LIN {X 0,Y 301.093,Z 516.104,A -85,B 0,C 180,E1 -16309.074,E2 -16309.074} C_VEL
LIN {X 0,Y 303.316,Z 506.78,A -85,B 0,C 180,E1 -16311.404,E2 -16311.404} C_VEL
LIN {X 0,Y 305.446,Z 497.307,A -85,B 0,C 180,E1 -16313.385,E2 -16313.385} C_VEL
LIN {X 0,Y 308.235,Z 485.037,A -85,B 0,C 180,E1 -16315.491,E2 -16315.491} C_VEL
LIN {X 0,Y 310.983,Z 472.541,A -85,B 0,C 180,E1 -16317.235,E2 -16317.235} C_VEL
LIN {X 0,Y 313.672,Z 459.222,A -85,B 0,C 180,E1 -16318.741,E2 -16318.741} C_VEL
LIN {X 0,Y 314.374,Z 455.035,A -85,B 0,C 180,E1 -16319.152,E2 -16319.152} C_VEL
LIN {X 0,Y 313.209,Z 443.277,A -85,B 0,C 180,E1 -16320.482,E2 -16320.482} C_VEL
LIN {X 0,Y 311.406,Z 431.077,A -85,B 0,C 180,E1 -16321.735,E2 -16321.735} C_VEL
LIN {X 0,Y 307.92,Z 415.559,A -85,B 0,C 180,E1 -16323.194,E2 -16323.194} C_VEL
LIN {X 0,Y 303.433,Z 400.922,A -85,B 0,C 180,E1 -16324.465,E2 -16324.465} C_VEL
LIN {X 0,Y 299.776,Z 390.786,A -85,B 0,C 180,E1 -16325.294,E2 -16325.294} C_VEL
LIN {X 0,Y 299.637,Z 389.858,A -85,B 0,C 180,E1 -16325.364,E2 -16325.364} C_VEL
LIN {X 0,Y 300.45,Z 384.591,A -85,B 0,C 180,E1 -16329.473,E2 -16329.473} C_VEL
LIN {X 0,Y 300.937,Z 380.64,A -85,B 0,C 180,E1 -16332.63,E2 -16332.63} C_VEL
LIN {X 0,Y 300.629,Z 377.385,A -85,B 0,C 180,E1 -16335.466,E2 -16335.466} C_VEL
LIN {X 0,Y 300.054,Z 373.593,A -85,B 0,C 180,E1 -16339.018,E2 -16339.018} C_VEL
LIN {X 0,Y 299.471,Z 370.212,A -85,B 0,C 180,E1 -16342.399,E2 -16342.399} C_VEL
LIN {X 0,Y 298.977,Z 367.207,A -85,B 0,C 180,E1 -16345.656,E2 -16345.656} C_VEL
LIN {X 0,Y 298.549,Z 364.477,A -85,B 0,C 180,E1 -16348.809,E2 -16348.809} C_VEL
LIN {X 0,Y 298.429,Z 363.938,A -85,B 0,C 180,E1 -16350.617,E2 -16350.617} C_VEL
LIN {X 0,Y 298.485,Z 363.932,A -85,B 0,C 180,E1 -16353.475,E2 -16353.475} C_VEL
LIN {X 0,Y 298.438,Z 363.938,A -85,B 0,C 180,E1 -16356.698,E2 -16356.698} C_VEL
LIN {X 0,Y 298.543,Z 363.922,A -85,B 0,C 180,E1 -16360.757,E2 -16360.757} C_VEL
LIN {X 0,Y 298.597,Z 363.92,A -85,B 0,C 180,E1 -16364.995,E2 -16364.995} C_VEL
LIN {X 0,Y 298.597,Z 363.922,A -85,B 0,C 180,E1 -16369.147,E2 -16369.147} C_VEL
LIN {X 0,Y 298.762,Z 363.898,A -85,B 0,C 180,E1 -16371.886,E2 -16371.886} C_VEL
LIN {X 0,Y 298.664,Z 363.908,A -85,B 0,C 180,E1 -16374.599,E2 -16374.599} C_VEL
LIN {X 0,Y 298.926,Z 363.874,A -85,B 0,C 180,E1 -16378.653,E2 -16378.653} C_VEL
LIN {X 0,Y 298.927,Z 363.876,A -85,B 0,C 180,E1 -16381.347,E2 -16381.347} C_VEL
LIN {X 0,Y 298.802,Z 363.885,A -85,B 0,C 180,E1 -16386.754,E2 -16386.754} C_VEL
LIN {X 0,Y 298.684,Z 363.904,A -85,B 0,C 180,E1 -16389.48,E2 -16389.48} C_VEL
LIN {X 0,Y 298.555,Z 363.892,A -85,B 0,C 180,E1 -16393.615,E2 -16393.615} C_VEL
LIN {X 0,Y 298.552,Z 363.921,A -85,B 0,C 180,E1 -16396.409,E2 -16396.409} C_VEL
LIN {X 0,Y 298.501,Z 363.902,A -85,B 0,C 180,E1 -16399.647,E2 -16399.647} C_VEL
LIN {X 0,Y 298.432,Z 363.935,A -85,B 0,C 180,E1 -16403.6,E2 -16403.6} C_VEL
LIN {X 0,Y 298.49,Z 363.909,A -85,B 0,C 180,E1 -16406.575,E2 -16406.575} C_VEL
LIN {X 0,Y 298.42,Z 363.936,A -85,B 0,C 180,E1 -16409.641,E2 -16409.641} C_VEL
LIN {X 0,Y 298.398,Z 363.924,A -85,B 0,C 180,E1 -16412.8,E2 -16412.8} C_VEL
LIN {X 0,Y 298.467,Z 363.933,A -85,B 0,C 180,E1 -16416.812,E2 -16416.812} C_VEL
LIN {X 0,Y 298.39,Z 363.942,A -85,B 0,C 180,E1 -16421.087,E2 -16421.087} C_VEL
LIN {X 0,Y 298.401,Z 363.942,A -85,B 0,C 180,E1 -16423.103,E2 -16423.103} C_VEL
LIN {X 0,Y 298.341,Z 363.954,A -85,B 0,C 180,E1 -16426.909,E2 -16426.909} C_VEL
LIN {X 0,Y 298.249,Z 363.963,A -85,B 0,C 180,E1 -16428.943,E2 -16428.943} C_VEL
LIN {X 0,Y 298.148,Z 365.832,A -85,B 0,C 180,E1 -16432.202,E2 -16432.202} C_VEL
LIN {X 0,Y 298.084,Z 367.347,A -85,B 0,C 180,E1 -16434.524,E2 -16434.524} C_VEL
LIN {X 0,Y 299.159,Z 370.435,A -85,B 0,C 180,E1 -16434.787,E2 -16434.787} C_VEL
LIN {X 0,Y 300.414,Z 372.767,A -85,B 0,C 180,E1 -16435.038,E2 -16435.038} C_VEL
LIN {X 0,Y 305.803,Z 384.256,A -85,B 0,C 180,E1 -16436.253,E2 -16436.253} C_VEL
LIN {X 0,Y 310.82,Z 397.125,A -85,B 0,C 180,E1 -16437.646,E2 -16437.646} C_VEL
LIN {X 0,Y 314.659,Z 409.849,A -85,B 0,C 180,E1 -16439.088,E2 -16439.088} C_VEL
LIN {X 0,Y 317.153,Z 421.115,A -85,B 0,C 180,E1 -16440.431,E2 -16440.431} C_VEL
LIN {X 0,Y 314.958,Z 434.259,A -85,B 0,C 180,E1 -16441.694,E2 -16441.694} C_VEL
LIN {X 0,Y 312.497,Z 447.415,A -85,B 0,C 180,E1 -16443.269,E2 -16443.269} C_VEL
LIN {X 0,Y 310.041,Z 458.721,A -85,B 0,C 180,E1 -16444.902,E2 -16444.902} C_VEL
LIN {X 0,Y 307.626,Z 469.495,A -85,B 0,C 180,E1 -16446.79,E2 -16446.79} C_VEL
LIN {X 0,Y 305.011,Z 480.245,A -85,B 0,C 180,E1 -16449.074,E2 -16449.074} C_VEL
LIN {X 0,Y 302.818,Z 489.159,A -85,B 0,C 180,E1 -16451.39,E2 -16451.39} C_VEL
LIN {X 0,Y 301.057,Z 496.534,A -85,B 0,C 180,E1 -16453.731,E2 -16453.731} C_VEL
LIN {X 0,Y 299.789,Z 501.835,A -85,B 0,C 180,E1 -16455.749,E2 -16455.749} C_VEL
LIN {X 0,Y 298.494,Z 507.611,A -85,B 0,C 180,E1 -16458.455,E2 -16458.455} C_VEL
LIN {X 0,Y 297.82,Z 511.025,A -85,B 0,C 180,E1 -16460.491,E2 -16460.491} C_VEL
LIN {X 0,Y 297.207,Z 514.571,A -85,B 0,C 180,E1 -16463.299,E2 -16463.299} C_VEL
LIN {X 0,Y 296.882,Z 516.759,A -85,B 0,C 180,E1 -16465.927,E2 -16465.927} C_VEL
LIN {X 0,Y 296.726,Z 517.922,A -85,B 0,C 180,E1 -16468.642,E2 -16468.642} C_VEL
LIN {X 0,Y 296.726,Z 517.935,A -85,B 0,C 180,E1 -16471.357,E2 -16471.357} C_VEL
LIN {X 0,Y 296.881,Z 516.827,A -85,B 0,C 180,E1 -16474.072,E2 -16474.072} C_VEL
LIN {X 0,Y 297.22,Z 514.599,A -85,B 0,C 180,E1 -16476.789,E2 -16476.789} C_VEL
LIN {X 0,Y 297.8,Z 511.195,A -85,B 0,C 180,E1 -16479.508,E2 -16479.508} C_VEL
LIN {X 0,Y 298.741,Z 506.528,A -85,B 0,C 180,E1 -16482.223,E2 -16482.223} C_VEL
LIN {X 0,Y 300.182,Z 500.468,A -85,B 0,C 180,E1 -16484.923,E2 -16484.923} C_VEL
LIN {X 0,Y 301.908,Z 492.838,A -85,B 0,C 180,E1 -16487.615,E2 -16487.615} C_VEL
LIN {X 0,Y 303.968,Z 484.686,A -85,B 0,C 180,E1 -16489.939,E2 -16489.939} C_VEL
LIN {X 0,Y 306.359,Z 474.857,A -85,B 0,C 180,E1 -16492.241,E2 -16492.241} C_VEL
LIN {X 0,Y 308.851,Z 464.107,A -85,B 0,C 180,E1 -16494.313,E2 -16494.313} C_VEL
LIN {X 0,Y 311.593,Z 451.648,A -85,B 0,C 180,E1 -16496.272,E2 -16496.272} C_VEL
LIN {X 0,Y 314.095,Z 439.396,A -85,B 0,C 180,E1 -16497.845,E2 -16497.845} C_VEL
LIN {X 0,Y 316.491,Z 425.99,A -85,B 0,C 180,E1 -16499.243,E2 -16499.243} C_VEL
LIN {X 0,Y 317.131,Z 420.255,A -85,B 0,C 180,E1 -16499.778,E2 -16499.778} C_VEL
LIN {X 0,Y 313.848,Z 406.769,A -85,B 0,C 180,E1 -16501.38,E2 -16501.38} C_VEL
LIN {X 0,Y 309.302,Z 392.975,A -85,B 0,C 180,E1 -16502.922,E2 -16502.922} C_VEL
LIN {X 0,Y 304.052,Z 380.298,A -85,B 0,C 180,E1 -16504.287,E2 -16504.287} C_VEL
LIN {X 0,Y 299.306,Z 370.651,A -85,B 0,C 180,E1 -16505.308,E2 -16505.308} C_VEL
LIN {X 0,Y 298.144,Z 367.656,A -85,B 0,C 180,E1 -16505.572,E2 -16505.572} C_VEL
LIN {X 0,Y 298.082,Z 367.317,A -85,B 0,C 180,E1 -16505.633,E2 -16505.633} C_VEL
LIN {X 0,Y 298.21,Z 364.814,A -85,B 0,C 180,E1 -16509.517,E2 -16509.517} C_VEL
LIN {X 0,Y 298.257,Z 363.953,A -85,B 0,C 180,E1 -16511.282,E2 -16511.282} C_VEL
LIN {X 0,Y 298.352,Z 363.946,A -85,B 0,C 180,E1 -16515.034,E2 -16515.034} C_VEL
LIN {X 0,Y 298.383,Z 363.944,A -85,B 0,C 180,E1 -16518.738,E2 -16518.738} C_VEL
LIN {X 0,Y 298.43,Z 363.938,A -85,B 0,C 180,E1 -16522.244,E2 -16522.244} C_VEL
LIN {X 0,Y 298.407,Z 363.933,A -85,B 0,C 180,E1 -16525.581,E2 -16525.581} C_VEL
LIN {X 0,Y 298.394,Z 363.938,A -85,B 0,C 180,E1 -16528.791,E2 -16528.791} C_VEL
LIN {X 0,Y 298.462,Z 363.917,A -85,B 0,C 180,E1 -16531.904,E2 -16531.904} C_VEL
LIN {X 0,Y 298.484,Z 363.925,A -85,B 0,C 180,E1 -16534.924,E2 -16534.924} C_VEL
LIN {X 0,Y 298.447,Z 363.908,A -85,B 0,C 180,E1 -16539.315,E2 -16539.315} C_VEL
LIN {X 0,Y 298.536,Z 363.92,A -85,B 0,C 180,E1 -16542.179,E2 -16542.179} C_VEL
LIN {X 0,Y 298.591,Z 363.905,A -85,B 0,C 180,E1 -16544.994,E2 -16544.994} C_VEL
LIN {X 0,Y 298.55,Z 363.895,A -85,B 0,C 180,E1 -16546.352,E2 -16546.352} C_VEL
LIN {X 0,Y 297.926,Z 363.976,A -85,B 0,C 180,E1 -16547.479,E2 -16547.479} C_VEL
LIN {X 0,Y 295.141,Z 364.34,A -85,B 0,C 180,E1 -16549.316,E2 -16549.316} C_VEL
LIN {X 0,Y 292.774,Z 364.642,A -85,B 0,C 180,E1 -16550.807,E2 -16550.807} C_VEL
LIN {X 0,Y 291.775,Z 364.763,A -85,B 0,C 180,E1 -16551.96,E2 -16551.96} C_VEL
LIN {X 0,Y 291.703,Z 364.771,A -85,B 0,C 180,E1 -16552.351,E2 -16552.351} C_VEL
LIN {X 0,Y 291.788,Z 364.767,A -85,B 0,C 180,E1 -16557.239,E2 -16557.239} C_VEL
LIN {X 0,Y 291.977,Z 364.743,A -85,B 0,C 180,E1 -16560,E2 -16560} C_VEL
LIN {X 0,Y 291.789,Z 364.764,A -85,B 0,C 180,E1 -16562.761,E2 -16562.761} C_VEL
LIN {X 0,Y 291.744,Z 364.77,A -85,B 0,C 180,E1 -16566.918,E2 -16566.918} C_VEL
LIN {X 0,Y 291.627,Z 364.784,A -85,B 0,C 180,E1 -16569.712,E2 -16569.712} C_VEL
LIN {X 0,Y 291.519,Z 364.798,A -85,B 0,C 180,E1 -16573.95,E2 -16573.95} C_VEL
LIN {X 0,Y 291.485,Z 364.801,A -85,B 0,C 180,E1 -16576.818,E2 -16576.818} C_VEL
LIN {X 0,Y 291.448,Z 364.807,A -85,B 0,C 180,E1 -16579.875,E2 -16579.875} C_VEL
LIN {X 0,Y 291.398,Z 364.816,A -85,B 0,C 180,E1 -16584.205,E2 -16584.205} C_VEL
LIN {X 0,Y 291.42,Z 364.813,A -85,B 0,C 180,E1 -16587.272,E2 -16587.272} C_VEL
LIN {X 0,Y 291.385,Z 364.86,A -85,B 0,C 180,E1 -16589.74,E2 -16589.74} C_VEL
LIN {X 0,Y 291.902,Z 368.045,A -85,B 0,C 180,E1 -16593.625,E2 -16593.625} C_VEL
LIN {X 0,Y 292.474,Z 371.514,A -85,B 0,C 180,E1 -16597.537,E2 -16597.537} C_VEL
LIN {X 0,Y 292.975,Z 374.262,A -85,B 0,C 180,E1 -16600.367,E2 -16600.367} C_VEL
LIN {X 0,Y 293.546,Z 378.133,A -85,B 0,C 180,E1 -16604.091,E2 -16604.091} C_VEL
LIN {X 0,Y 293.914,Z 381.424,A -85,B 0,C 180,E1 -16607.042,E2 -16607.042} C_VEL
LIN {X 0,Y 293.528,Z 384.953,A -85,B 0,C 180,E1 -16610.012,E2 -16610.012} C_VEL
LIN {X 0,Y 292.75,Z 389.496,A -85,B 0,C 180,E1 -16613.667,E2 -16613.667} C_VEL
LIN {X 0,Y 293.745,Z 392.872,A -85,B 0,C 180,E1 -16613.917,E2 -16613.917} C_VEL
LIN {X 0,Y 298.154,Z 404.831,A -85,B 0,C 180,E1 -16614.994,E2 -16614.994} C_VEL
LIN {X 0,Y 302.141,Z 418.676,A -85,B 0,C 180,E1 -16616.283,E2 -16616.283} C_VEL
LIN {X 0,Y 305.296,Z 433.414,A -85,B 0,C 180,E1 -16617.756,E2 -16617.756} C_VEL
LIN {X 0,Y 307.228,Z 447.699,A -85,B 0,C 180,E1 -16619.314,E2 -16619.314} C_VEL
LIN {X 0,Y 307.893,Z 456.22,A -85,B 0,C 180,E1 -16620.329,E2 -16620.329} C_VEL
LIN {X 0,Y 305.201,Z 469.763,A -85,B 0,C 180,E1 -16621.832,E2 -16621.832} C_VEL
LIN {X 0,Y 302.549,Z 481.597,A -85,B 0,C 180,E1 -16623.439,E2 -16623.439} C_VEL
LIN {X 0,Y 300.146,Z 491.697,A -85,B 0,C 180,E1 -16625.073,E2 -16625.073} C_VEL
LIN {X 0,Y 297.432,Z 502.993,A -85,B 0,C 180,E1 -16627.292,E2 -16627.292} C_VEL
LIN {X 0,Y 295.325,Z 512.081,A -85,B 0,C 180,E1 -16629.451,E2 -16629.451} C_VEL
LIN {X 0,Y 293.288,Z 520.461,A -85,B 0,C 180,E1 -16631.85,E2 -16631.85} C_VEL
LIN {X 0,Y 291.593,Z 528.35,A -85,B 0,C 180,E1 -16634.626,E2 -16634.626} C_VEL
LIN {X 0,Y 290.489,Z 534.643,A -85,B 0,C 180,E1 -16637.424,E2 -16637.424} C_VEL
LIN {X 0,Y 289.783,Z 539.519,A -85,B 0,C 180,E1 -16640.226,E2 -16640.226} C_VEL
LIN {X 0,Y 289.55,Z 543.105,A -85,B 0,C 180,E1 -16643.03,E2 -16643.03} C_VEL
LIN {X 0,Y 289.515,Z 545.468,A -85,B 0,C 180,E1 -16645.824,E2 -16645.824} C_VEL
LIN {X 0,Y 289.53,Z 546.656,A -85,B 0,C 180,E1 -16648.61,E2 -16648.61} C_VEL
LIN {X 0,Y 289.581,Z 546.815,A -85,B 0,C 180,E1 -16650.001,E2 -16650.001} C_VEL
LIN {X 0,Y 289.524,Z 546.197,A -85,B 0,C 180,E1 -16652.783,E2 -16652.783} C_VEL
LIN {X 0,Y 289.586,Z 544.299,A -85,B 0,C 180,E1 -16655.713,E2 -16655.713} C_VEL
LIN {X 0,Y 289.627,Z 541.438,A -85,B 0,C 180,E1 -16658.372,E2 -16658.372} C_VEL
LIN {X 0,Y 290.039,Z 537.211,A -85,B 0,C 180,E1 -16661.178,E2 -16661.178} C_VEL
LIN {X 0,Y 290.979,Z 531.633,A -85,B 0,C 180,E1 -16663.977,E2 -16663.977} C_VEL
LIN {X 0,Y 292.401,Z 524.549,A -85,B 0,C 180,E1 -16666.764,E2 -16666.764} C_VEL
LIN {X 0,Y 294.312,Z 515.75,A -85,B 0,C 180,E1 -16669.531,E2 -16669.531} C_VEL
LIN {X 0,Y 296.621,Z 506.425,A -85,B 0,C 180,E1 -16671.912,E2 -16671.912} C_VEL
LIN {X 0,Y 298.867,Z 496.952,A -85,B 0,C 180,E1 -16673.932,E2 -16673.932} C_VEL
LIN {X 0,Y 301.779,Z 484.683,A -85,B 0,C 180,E1 -16676.077,E2 -16676.077} C_VEL
LIN {X 0,Y 304.616,Z 472.185,A -85,B 0,C 180,E1 -16677.853,E2 -16677.853} C_VEL
LIN {X 0,Y 307.466,Z 458.73,A -85,B 0,C 180,E1 -16679.394,E2 -16679.394} C_VEL
LIN {X 0,Y 307.877,Z 456.13,A -85,B 0,C 180,E1 -16679.657,E2 -16679.657} C_VEL
LIN {X 0,Y 306.607,Z 442.894,A -85,B 0,C 180,E1 -16681.211,E2 -16681.211} C_VEL
LIN {X 0,Y 304.714,Z 430.324,A -85,B 0,C 180,E1 -16682.546,E2 -16682.546} C_VEL
LIN {X 0,Y 301.144,Z 414.784,A -85,B 0,C 180,E1 -16684.064,E2 -16684.064} C_VEL
LIN {X 0,Y 296.174,Z 399.218,A -85,B 0,C 180,E1 -16685.491,E2 -16685.491} C_VEL
LIN {X 0,Y 293.567,Z 392.489,A -85,B 0,C 180,E1 -16686.087,E2 -16686.087} C_VEL
LIN {X 0,Y 292.771,Z 389.434,A -85,B 0,C 180,E1 -16686.339,E2 -16686.339} C_VEL
LIN {X 0,Y 293.539,Z 384.573,A -85,B 0,C 180,E1 -16690.275,E2 -16690.275} C_VEL
LIN {X 0,Y 293.915,Z 381.328,A -85,B 0,C 180,E1 -16692.959,E2 -16692.959} C_VEL
LIN {X 0,Y 293.53,Z 377.943,A -85,B 0,C 180,E1 -16696.025,E2 -16696.025} C_VEL
LIN {X 0,Y 292.945,Z 374.215,A -85,B 0,C 180,E1 -16699.628,E2 -16699.628} C_VEL
LIN {X 0,Y 292.427,Z 370.907,A -85,B 0,C 180,E1 -16703.071,E2 -16703.071} C_VEL
LIN {X 0,Y 291.874,Z 367.974,A -85,B 0,C 180,E1 -16706.371,E2 -16706.371} C_VEL
LIN {X 0,Y 291.386,Z 364.816,A -85,B 0,C 180,E1 -16710.262,E2 -16710.262} C_VEL
LIN {X 0,Y 291.419,Z 364.812,A -85,B 0,C 180,E1 -16714.272,E2 -16714.272} C_VEL
LIN {X 0,Y 291.385,Z 364.815,A -85,B 0,C 180,E1 -16717.3,E2 -16717.3} C_VEL
LIN {X 0,Y 291.462,Z 364.806,A -85,B 0,C 180,E1 -16720.271,E2 -16720.271} C_VEL
LIN {X 0,Y 291.558,Z 364.796,A -85,B 0,C 180,E1 -16724.624,E2 -16724.624} C_VEL
LIN {X 0,Y 291.54,Z 364.799,A -85,B 0,C 180,E1 -16728.881,E2 -16728.881} C_VEL
LIN {X 0,Y 291.713,Z 364.776,A -85,B 0,C 180,E1 -16731.689,E2 -16731.689} C_VEL
LIN {X 0,Y 291.634,Z 364.784,A -85,B 0,C 180,E1 -16734.469,E2 -16734.469} C_VEL
LIN {X 0,Y 291.892,Z 364.751,A -85,B 0,C 180,E1 -16738.62,E2 -16738.62} C_VEL
LIN {X 0,Y 291.894,Z 364.753,A -85,B 0,C 180,E1 -16741.38,E2 -16741.38} C_VEL
LIN {X 0,Y 291.75,Z 364.763,A -85,B 0,C 180,E1 -16746.918,E2 -16746.918} C_VEL
LIN {X 0,Y 291.633,Z 364.782,A -85,B 0,C 180,E1 -16749.712,E2 -16749.712} C_VEL
LIN {X 0,Y 291.525,Z 364.771,A -85,B 0,C 180,E1 -16753.95,E2 -16753.95} C_VEL
LIN {X 0,Y 291.49,Z 364.801,A -85,B 0,C 180,E1 -16756.818,E2 -16756.818} C_VEL
LIN {X 0,Y 291.454,Z 364.777,A -85,B 0,C 180,E1 -16759.875,E2 -16759.875} C_VEL
LIN {X 0,Y 291.387,Z 364.814,A -85,B 0,C 180,E1 -16764.207,E2 -16764.207} C_VEL
LIN {X 0,Y 291.423,Z 364.786,A -85,B 0,C 180,E1 -16767.272,E2 -16767.272} C_VEL
LIN {X 0,Y 291.337,Z 364.821,A -85,B 0,C 180,E1 -16770.437,E2 -16770.437} C_VEL
LIN {X 0,Y 291.348,Z 364.8,A -85,B 0,C 180,E1 -16773.698,E2 -16773.698} C_VEL
LIN {X 0,Y 291.397,Z 364.813,A -85,B 0,C 180,E1 -16777.258,E2 -16777.258} C_VEL
LIN {X 0,Y 291.337,Z 364.823,A -85,B 0,C 180,E1 -16780.642,E2 -16780.642} C_VEL
LIN {X 0,Y 291.293,Z 364.829,A -85,B 0,C 180,E1 -16784.402,E2 -16784.402} C_VEL
LIN {X 0,Y 291.218,Z 364.84,A -85,B 0,C 180,E1 -16788.429,E2 -16788.429} C_VEL
LIN {X 0,Y 291.195,Z 366.217,A -85,B 0,C 180,E1 -16791.133,E2 -16791.133} C_VEL
LIN {X 0,Y 291.077,Z 367.767,A -85,B 0,C 180,E1 -16793.544,E2 -16793.544} C_VEL
LIN {X 0,Y 292.155,Z 370.783,A -85,B 0,C 180,E1 -16793.808,E2 -16793.808} C_VEL
LIN {X 0,Y 293.526,Z 373.281,A -85,B 0,C 180,E1 -16794.095,E2 -16794.095} C_VEL
LIN {X 0,Y 299.644,Z 386.04,A -85,B 0,C 180,E1 -16795.541,E2 -16795.541} C_VEL
LIN {X 0,Y 304.505,Z 398.844,A -85,B 0,C 180,E1 -16796.99,E2 -16796.99} C_VEL
LIN {X 0,Y 308.201,Z 410.948,A -85,B 0,C 180,E1 -16798.428,E2 -16798.428} C_VEL
LIN {X 0,Y 310.796,Z 422.533,A -85,B 0,C 180,E1 -16799.877,E2 -16799.877} C_VEL
LIN {X 0,Y 308.47,Z 436.029,A -85,B 0,C 180,E1 -16801.229,E2 -16801.229} C_VEL
LIN {X 0,Y 305.911,Z 448.932,A -85,B 0,C 180,E1 -16802.831,E2 -16802.831} C_VEL
LIN {X 0,Y 303.238,Z 460.593,A -85,B 0,C 180,E1 -16804.588,E2 -16804.588} C_VEL
LIN {X 0,Y 300.657,Z 471.474,A -85,B 0,C 180,E1 -16806.585,E2 -16806.585} C_VEL
LIN {X 0,Y 298.369,Z 480.597,A -85,B 0,C 180,E1 -16808.586,E2 -16808.586} C_VEL
LIN {X 0,Y 296.077,Z 489.51,A -85,B 0,C 180,E1 -16810.95,E2 -16810.95} C_VEL
LIN {X 0,Y 294.19,Z 496.887,A -85,B 0,C 180,E1 -16813.341,E2 -16813.341} C_VEL
LIN {X 0,Y 292.903,Z 502.185,A -85,B 0,C 180,E1 -16815.407,E2 -16815.407} C_VEL
LIN {X 0,Y 291.536,Z 507.96,A -85,B 0,C 180,E1 -16818.175,E2 -16818.175} C_VEL
LIN {X 0,Y 290.826,Z 511.373,A -85,B 0,C 180,E1 -16820.26,E2 -16820.26} C_VEL
LIN {X 0,Y 290.136,Z 515.078,A -85,B 0,C 180,E1 -16823.291,E2 -16823.291} C_VEL
LIN {X 0,Y 289.821,Z 517.106,A -85,B 0,C 180,E1 -16825.828,E2 -16825.828} C_VEL
LIN {X 0,Y 289.639,Z 518.269,A -85,B 0,C 180,E1 -16828.609,E2 -16828.609} C_VEL
LIN {X 0,Y 289.639,Z 518.283,A -85,B 0,C 180,E1 -16831.39,E2 -16831.39} C_VEL
LIN {X 0,Y 289.82,Z 517.174,A -85,B 0,C 180,E1 -16834.171,E2 -16834.171} C_VEL
LIN {X 0,Y 290.165,Z 514.947,A -85,B 0,C 180,E1 -16836.955,E2 -16836.955} C_VEL
LIN {X 0,Y 290.804,Z 511.542,A -85,B 0,C 180,E1 -16839.739,E2 -16839.739} C_VEL
LIN {X 0,Y 291.796,Z 506.875,A -85,B 0,C 180,E1 -16842.519,E2 -16842.519} C_VEL
LIN {X 0,Y 293.291,Z 500.816,A -85,B 0,C 180,E1 -16845.282,E2 -16845.282} C_VEL
LIN {X 0,Y 295.123,Z 493.185,A -85,B 0,C 180,E1 -16848.033,E2 -16848.033} C_VEL
LIN {X 0,Y 297.278,Z 485.033,A -85,B 0,C 180,E1 -16850.408,E2 -16850.408} C_VEL
LIN {X 0,Y 299.778,Z 475.204,A -85,B 0,C 180,E1 -16852.756,E2 -16852.756} C_VEL
LIN {X 0,Y 302.488,Z 464.055,A -85,B 0,C 180,E1 -16854.936,E2 -16854.936} C_VEL
LIN {X 0,Y 305.233,Z 451.993,A -85,B 0,C 180,E1 -16856.863,E2 -16856.863} C_VEL
LIN {X 0,Y 307.842,Z 439.739,A -85,B 0,C 180,E1 -16858.461,E2 -16858.461} C_VEL
LIN {X 0,Y 310.329,Z 426.332,A -85,B 0,C 180,E1 -16859.882,E2 -16859.882} C_VEL
LIN {X 0,Y 310.808,Z 423.045,A -85,B 0,C 180,E1 -16860.185,E2 -16860.185} C_VEL
LIN {X 0,Y 309.093,Z 414.317,A -85,B 0,C 180,E1 -16861.27,E2 -16861.27} C_VEL
LIN {X 0,Y 305.722,Z 402.495,A -85,B 0,C 180,E1 -16862.697,E2 -16862.697} C_VEL
LIN {X 0,Y 301.143,Z 389.817,A -85,B 0,C 180,E1 -16864.169,E2 -16864.169} C_VEL
LIN {X 0,Y 295.84,Z 377.893,A -85,B 0,C 180,E1 -16865.511,E2 -16865.511} C_VEL
LIN {X 0,Y 292.558,Z 371.39,A -85,B 0,C 180,E1 -16866.237,E2 -16866.237} C_VEL
LIN {X 0,Y 291.302,Z 368.749,A -85,B 0,C 180,E1 -16866.516,E2 -16866.516} C_VEL
LIN {X 0,Y 291.104,Z 367.725,A -85,B 0,C 180,E1 -16866.608,E2 -16866.608} C_VEL
LIN {X 0,Y 291.205,Z 365.953,A -85,B 0,C 180,E1 -16869.439,E2 -16869.439} C_VEL
LIN {X 0,Y 291.214,Z 364.83,A -85,B 0,C 180,E1 -16871.571,E2 -16871.571} C_VEL
LIN {X 0,Y 291.289,Z 364.826,A -85,B 0,C 180,E1 -16875.598,E2 -16875.598} C_VEL
LIN {X 0,Y 291.333,Z 364.821,A -85,B 0,C 180,E1 -16879.357,E2 -16879.357} C_VEL
LIN {X 0,Y 291.423,Z 364.809,A -85,B 0,C 180,E1 -16882.922,E2 -16882.922} C_VEL
LIN {X 0,Y 291.343,Z 364.804,A -85,B 0,C 180,E1 -16886.301,E2 -16886.301} C_VEL
LIN {X 0,Y 291.386,Z 364.813,A -85,B 0,C 180,E1 -16890.26,E2 -16890.26} C_VEL
LIN {X 0,Y 291.415,Z 364.798,A -85,B 0,C 180,E1 -16894.272,E2 -16894.272} C_VEL
LIN {X 0,Y 291.38,Z 364.809,A -85,B 0,C 180,E1 -16897.299,E2 -16897.299} C_VEL
LIN {X 0,Y 291.456,Z 364.781,A -85,B 0,C 180,E1 -16900.27,E2 -16900.27} C_VEL
LIN {X 0,Y 291.553,Z 364.785,A -85,B 0,C 180,E1 -16904.623,E2 -16904.623} C_VEL
LIN {X 0,Y 291.537,Z 364.785,A -85,B 0,C 180,E1 -16908.88,E2 -16908.88} C_VEL
LIN {X 0,Y 291.703,Z 364.771,A -85,B 0,C 180,E1 -16912.351,E2 -16912.351} C_VEL
LIN {X 0,Y 291.053,Z 364.856,A -85,B 0,C 180,E1 -16913.502,E2 -16913.502} C_VEL
LIN {X 0,Y 288.196,Z 365.213,A -85,B 0,C 180,E1 -16915.376,E2 -16915.376} C_VEL
LIN {X 0,Y 285.817,Z 365.508,A -85,B 0,C 180,E1 -16916.898,E2 -16916.898} C_VEL
LIN {X 0,Y 284.873,Z 365.626,A -85,B 0,C 180,E1 -16918.077,E2 -16918.077} C_VEL
LIN {X 0,Y 284.839,Z 365.629,A -85,B 0,C 180,E1 -16918.476,E2 -16918.476} C_VEL
LIN {X 0,Y 284.854,Z 365.63,A -85,B 0,C 180,E1 -16921.414,E2 -16921.414} C_VEL
LIN {X 0,Y 284.696,Z 365.648,A -85,B 0,C 180,E1 -16927.09,E2 -16927.09} C_VEL
LIN {X 0,Y 284.564,Z 365.663,A -85,B 0,C 180,E1 -16929.955,E2 -16929.955} C_VEL
LIN {X 0,Y 284.479,Z 365.674,A -85,B 0,C 180,E1 -16934.303,E2 -16934.303} C_VEL
LIN {X 0,Y 284.423,Z 365.681,A -85,B 0,C 180,E1 -16937.248,E2 -16937.248} C_VEL
LIN {X 0,Y 284.376,Z 365.685,A -85,B 0,C 180,E1 -16940.242,E2 -16940.242} C_VEL
LIN {X 0,Y 284.367,Z 365.691,A -85,B 0,C 180,E1 -16943.876,E2 -16943.876} C_VEL
LIN {X 0,Y 284.395,Z 365.688,A -85,B 0,C 180,E1 -16947.174,E2 -16947.174} C_VEL
LIN {X 0,Y 284.417,Z 366.236,A -85,B 0,C 180,E1 -16949.617,E2 -16949.617} C_VEL
LIN {X 0,Y 284.845,Z 368.875,A -85,B 0,C 180,E1 -16952.979,E2 -16952.979} C_VEL
LIN {X 0,Y 285.307,Z 371.683,A -85,B 0,C 180,E1 -16956.242,E2 -16956.242} C_VEL
LIN {X 0,Y 285.987,Z 375.526,A -85,B 0,C 180,E1 -16960.377,E2 -16960.377} C_VEL
LIN {X 0,Y 286.601,Z 379.899,A -85,B 0,C 180,E1 -16964.674,E2 -16964.674} C_VEL
LIN {X 0,Y 286.865,Z 382.78,A -85,B 0,C 180,E1 -16967.305,E2 -16967.305} C_VEL
LIN {X 0,Y 286.389,Z 386.32,A -85,B 0,C 180,E1 -16970.355,E2 -16970.355} C_VEL
LIN {X 0,Y 285.918,Z 389.064,A -85,B 0,C 180,E1 -16972.637,E2 -16972.637} C_VEL
LIN {X 0,Y 286.878,Z 392.47,A -85,B 0,C 180,E1 -16972.911,E2 -16972.911} C_VEL
LIN {X 0,Y 287.832,Z 394.8,A -85,B 0,C 180,E1 -16973.136,E2 -16973.136} C_VEL
LIN {X 0,Y 292.175,Z 406.787,A -85,B 0,C 180,E1 -16974.278,E2 -16974.278} C_VEL
LIN {X 0,Y 296.225,Z 421.176,A -85,B 0,C 180,E1 -16975.706,E2 -16975.706} C_VEL
LIN {X 0,Y 299.257,Z 436.303,A -85,B 0,C 180,E1 -16977.307,E2 -16977.307} C_VEL
LIN {X 0,Y 300.89,Z 449.869,A -85,B 0,C 180,E1 -16978.871,E2 -16978.871} C_VEL
LIN {X 0,Y 301.417,Z 457.273,A -85,B 0,C 180,E1 -16979.796,E2 -16979.796} C_VEL
LIN {X 0,Y 298.926,Z 469.417,A -85,B 0,C 180,E1 -16981.186,E2 -16981.186} C_VEL
LIN {X 0,Y 295.9,Z 482.326,A -85,B 0,C 180,E1 -16982.984,E2 -16982.984} C_VEL
LIN {X 0,Y 293.193,Z 493.145,A -85,B 0,C 180,E1 -16984.82,E2 -16984.82} C_VEL
LIN {X 0,Y 290.642,Z 503.338,A -85,B 0,C 180,E1 -16986.905,E2 -16986.905} C_VEL
LIN {X 0,Y 288.622,Z 511.731,A -85,B 0,C 180,E1 -16988.952,E2 -16988.952} C_VEL
LIN {X 0,Y 286.463,Z 520.11,A -85,B 0,C 180,E1 -16991.402,E2 -16991.402} C_VEL
LIN {X 0,Y 284.627,Z 528.303,A -85,B 0,C 180,E1 -16994.362,E2 -16994.362} C_VEL
LIN {X 0,Y 283.495,Z 534.293,A -85,B 0,C 180,E1 -16997.109,E2 -16997.109} C_VEL
LIN {X 0,Y 282.73,Z 539.169,A -85,B 0,C 180,E1 -16999.98,E2 -16999.98} C_VEL
LIN {X 0,Y 282.465,Z 542.755,A -85,B 0,C 180,E1 -17002.854,E2 -17002.854} C_VEL
LIN {X 0,Y 282.415,Z 545.119,A -85,B 0,C 180,E1 -17005.719,E2 -17005.719} C_VEL
LIN {X 0,Y 282.447,Z 546.309,A -85,B 0,C 180,E1 -17008.575,E2 -17008.575} C_VEL
LIN {X 0,Y 282.494,Z 546.467,A -85,B 0,C 180,E1 -17010.001,E2 -17010.001} C_VEL
LIN {X 0,Y 282.45,Z 545.85,A -85,B 0,C 180,E1 -17012.853,E2 -17012.853} C_VEL
LIN {X 0,Y 282.487,Z 544.067,A -85,B 0,C 180,E1 -17015.712,E2 -17015.712} C_VEL
LIN {X 0,Y 282.557,Z 541.087,A -85,B 0,C 180,E1 -17018.583,E2 -17018.583} C_VEL
LIN {X 0,Y 283.011,Z 536.859,A -85,B 0,C 180,E1 -17021.459,E2 -17021.459} C_VEL
LIN {X 0,Y 284.02,Z 531.28,A -85,B 0,C 180,E1 -17024.327,E2 -17024.327} C_VEL
LIN {X 0,Y 285.519,Z 524.195,A -85,B 0,C 180,E1 -17027.181,E2 -17027.181} C_VEL
LIN {X 0,Y 287.555,Z 515.396,A -85,B 0,C 180,E1 -17030.01,E2 -17030.01} C_VEL
LIN {X 0,Y 289.96,Z 506.07,A -85,B 0,C 180,E1 -17032.442,E2 -17032.442} C_VEL
LIN {X 0,Y 292.334,Z 496.599,A -85,B 0,C 180,E1 -17034.502,E2 -17034.502} C_VEL
LIN {X 0,Y 295.357,Z 484.328,A -85,B 0,C 180,E1 -17036.688,E2 -17036.688} C_VEL
LIN {X 0,Y 298.345,Z 471.833,A -85,B 0,C 180,E1 -17038.492,E2 -17038.492} C_VEL
LIN {X 0,Y 301.005,Z 459.613,A -85,B 0,C 180,E1 -17039.931,E2 -17039.931} C_VEL
LIN {X 0,Y 301.351,Z 457.667,A -85,B 0,C 180,E1 -17040.136,E2 -17040.136} C_VEL
LIN {X 0,Y 300.396,Z 445.416,A -85,B 0,C 180,E1 -17041.642,E2 -17041.642} C_VEL
LIN {X 0,Y 298.493,Z 432.171,A -85,B 0,C 180,E1 -17043.117,E2 -17043.117} C_VEL
LIN {X 0,Y 295.244,Z 417.409,A -85,B 0,C 180,E1 -17044.642,E2 -17044.642} C_VEL
LIN {X 0,Y 290.815,Z 402.842,A -85,B 0,C 180,E1 -17046.063,E2 -17046.063} C_VEL
LIN {X 0,Y 287.082,Z 392.869,A -85,B 0,C 180,E1 -17047.008,E2 -17047.008} C_VEL
LIN {X 0,Y 286.001,Z 389.931,A -85,B 0,C 180,E1 -17047.271,E2 -17047.271} C_VEL
LIN {X 0,Y 285.911,Z 389.023,A -85,B 0,C 180,E1 -17047.366,E2 -17047.366} C_VEL
LIN {X 0,Y 286.756,Z 384.185,A -85,B 0,C 180,E1 -17051.433,E2 -17051.433} C_VEL
LIN {X 0,Y 286.885,Z 382.013,A -85,B 0,C 180,E1 -17053.31,E2 -17053.31} C_VEL
LIN {X 0,Y 286.406,Z 378.481,A -85,B 0,C 180,E1 -17056.601,E2 -17056.601} C_VEL
LIN {X 0,Y 285.867,Z 374.837,A -85,B 0,C 180,E1 -17060.268,E2 -17060.268} C_VEL
LIN {X 0,Y 285.218,Z 371.049,A -85,B 0,C 180,E1 -17064.406,E2 -17064.406} C_VEL
LIN {X 0,Y 284.588,Z 367.422,A -85,B 0,C 180,E1 -17068.762,E2 -17068.762} C_VEL
LIN {X 0,Y 284.415,Z 366.184,A -85,B 0,C 180,E1 -17070.383,E2 -17070.383} C_VEL
LIN {X 0,Y 284.399,Z 365.686,A -85,B 0,C 180,E1 -17072.827,E2 -17072.827} C_VEL
LIN {X 0,Y 284.369,Z 365.69,A -85,B 0,C 180,E1 -17076.707,E2 -17076.707} C_VEL
LIN {X 0,Y 284.407,Z 365.685,A -85,B 0,C 180,E1 -17081.262,E2 -17081.262} C_VEL
LIN {X 0,Y 284.495,Z 365.676,A -85,B 0,C 180,E1 -17084.459,E2 -17084.459} C_VEL
LIN {X 0,Y 284.492,Z 365.677,A -85,B 0,C 180,E1 -17088.602,E2 -17088.602} C_VEL
LIN {X 0,Y 284.663,Z 365.654,A -85,B 0,C 180,E1 -17091.481,E2 -17091.481} C_VEL
LIN {X 0,Y 284.605,Z 365.659,A -85,B 0,C 180,E1 -17094.331,E2 -17094.331} C_VEL
LIN {X 0,Y 284.858,Z 365.627,A -85,B 0,C 180,E1 -17098.586,E2 -17098.586} C_VEL
LIN {X 0,Y 284.86,Z 365.629,A -85,B 0,C 180,E1 -17101.414,E2 -17101.414} C_VEL
LIN {X 0,Y 284.702,Z 365.641,A -85,B 0,C 180,E1 -17107.09,E2 -17107.09} C_VEL
LIN {X 0,Y 284.57,Z 365.66,A -85,B 0,C 180,E1 -17109.955,E2 -17109.955} C_VEL
LIN {X 0,Y 284.485,Z 365.652,A -85,B 0,C 180,E1 -17114.303,E2 -17114.303} C_VEL
LIN {X 0,Y 284.427,Z 365.679,A -85,B 0,C 180,E1 -17117.248,E2 -17117.248} C_VEL
LIN {X 0,Y 284.381,Z 365.656,A -85,B 0,C 180,E1 -17120.242,E2 -17120.242} C_VEL
LIN {X 0,Y 284.341,Z 365.688,A -85,B 0,C 180,E1 -17124.846,E2 -17124.846} C_VEL
LIN {X 0,Y 284.331,Z 365.672,A -85,B 0,C 180,E1 -17128.011,E2 -17128.011} C_VEL
LIN {X 0,Y 284.297,Z 365.695,A -85,B 0,C 180,E1 -17131.274,E2 -17131.274} C_VEL
LIN {X 0,Y 284.365,Z 365.686,A -85,B 0,C 180,E1 -17135.354,E2 -17135.354} C_VEL
LIN {X 0,Y 284.326,Z 365.695,A -85,B 0,C 180,E1 -17138.167,E2 -17138.167} C_VEL
LIN {X 0,Y 284.272,Z 365.703,A -85,B 0,C 180,E1 -17142.124,E2 -17142.124} C_VEL
LIN {X 0,Y 284.22,Z 365.712,A -85,B 0,C 180,E1 -17146.182,E2 -17146.182} C_VEL
LIN {X 0,Y 284.175,Z 365.718,A -85,B 0,C 180,E1 -17148.106,E2 -17148.106} C_VEL
LIN {X 0,Y 284.169,Z 366.676,A -85,B 0,C 180,E1 -17150.057,E2 -17150.057} C_VEL
LIN {X 0,Y 284.079,Z 368.156,A -85,B 0,C 180,E1 -17152.477,E2 -17152.477} C_VEL
LIN {X 0,Y 285.229,Z 371.291,A -85,B 0,C 180,E1 -17152.786,E2 -17152.786} C_VEL
LIN {X 0,Y 286.426,Z 373.265,A -85,B 0,C 180,E1 -17153.043,E2 -17153.043} C_VEL
LIN {X 0,Y 292.526,Z 385.915,A -85,B 0,C 180,E1 -17154.546,E2 -17154.546} C_VEL
LIN {X 0,Y 297.068,Z 397.186,A -85,B 0,C 180,E1 -17155.897,E2 -17155.897} C_VEL
LIN {X 0,Y 301.193,Z 409.976,A -85,B 0,C 180,E1 -17157.482,E2 -17157.482} C_VEL
LIN {X 0,Y 304.121,Z 422.384,A -85,B 0,C 180,E1 -17159.085,E2 -17159.085} C_VEL
LIN {X 0,Y 304.468,Z 424.418,A -85,B 0,C 180,E1 -17159.351,E2 -17159.351} C_VEL
LIN {X 0,Y 302,Z 437.799,A -85,B 0,C 180,E1 -17160.744,E2 -17160.744} C_VEL
LIN {X 0,Y 299.332,Z 450.45,A -85,B 0,C 180,E1 -17162.373,E2 -17162.373} C_VEL
LIN {X 0,Y 296.4,Z 462.662,A -85,B 0,C 180,E1 -17164.293,E2 -17164.293} C_VEL
LIN {X 0,Y 293.727,Z 473.436,A -85,B 0,C 180,E1 -17166.373,E2 -17166.373} C_VEL
LIN {X 0,Y 291.027,Z 483.624,A -85,B 0,C 180,E1 -17168.762,E2 -17168.762} C_VEL
LIN {X 0,Y 288.731,Z 492.074,A -85,B 0,C 180,E1 -17171.184,E2 -17171.184} C_VEL
LIN {X 0,Y 286.921,Z 499.093,A -85,B 0,C 180,E1 -17173.638,E2 -17173.638} C_VEL
LIN {X 0,Y 285.199,Z 505.603,A -85,B 0,C 180,E1 -17176.461,E2 -17176.461} C_VEL
LIN {X 0,Y 284.076,Z 510.678,A -85,B 0,C 180,E1 -17179.306,E2 -17179.306} C_VEL
LIN {X 0,Y 283.386,Z 513.603,A -85,B 0,C 180,E1 -17181.442,E2 -17181.442} C_VEL
LIN {X 0,Y 282.91,Z 516.457,A -85,B 0,C 180,E1 -17184.297,E2 -17184.297} C_VEL
LIN {X 0,Y 282.624,Z 518.173,A -85,B 0,C 180,E1 -17187.149,E2 -17187.149} C_VEL
LIN {X 0,Y 282.541,Z 518.772,A -85,B 0,C 180,E1 -17189.999,E2 -17189.999} C_VEL
LIN {X 0,Y 282.624,Z 518.213,A -85,B 0,C 180,E1 -17192.85,E2 -17192.85} C_VEL
LIN {X 0,Y 282.912,Z 516.55,A -85,B 0,C 180,E1 -17195.702,E2 -17195.702} C_VEL
LIN {X 0,Y 283.381,Z 513.745,A -85,B 0,C 180,E1 -17198.557,E2 -17198.557} C_VEL
LIN {X 0,Y 284.254,Z 509.721,A -85,B 0,C 180,E1 -17201.407,E2 -17201.407} C_VEL
LIN {X 0,Y 285.499,Z 504.381,A -85,B 0,C 180,E1 -17204.25,E2 -17204.25} C_VEL
LIN {X 0,Y 286.889,Z 499.382,A -85,B 0,C 180,E1 -17206.362,E2 -17206.362} C_VEL
LIN {X 0,Y 288.633,Z 492.431,A -85,B 0,C 180,E1 -17208.821,E2 -17208.821} C_VEL
LIN {X 0,Y 290.96,Z 484.047,A -85,B 0,C 180,E1 -17211.242,E2 -17211.242} C_VEL
LIN {X 0,Y 293.621,Z 473.945,A -85,B 0,C 180,E1 -17213.635,E2 -17213.635} C_VEL
LIN {X 0,Y 296.462,Z 462.732,A -85,B 0,C 180,E1 -17215.803,E2 -17215.803} C_VEL
LIN {X 0,Y 299.193,Z 451.171,A -85,B 0,C 180,E1 -17217.64,E2 -17217.64} C_VEL
LIN {X 0,Y 301.609,Z 440.083,A -85,B 0,C 180,E1 -17219.105,E2 -17219.105} C_VEL
LIN {X 0,Y 304.194,Z 426.674,A -85,B 0,C 180,E1 -17220.549,E2 -17220.549} C_VEL
LIN {X 0,Y 304.495,Z 424.172,A -85,B 0,C 180,E1 -17220.792,E2 -17220.792} C_VEL
LIN {X 0,Y 301.751,Z 411.982,A -85,B 0,C 180,E1 -17222.39,E2 -17222.39} C_VEL
LIN {X 0,Y 297.823,Z 399.308,A -85,B 0,C 180,E1 -17223.966,E2 -17223.966} C_VEL
LIN {X 0,Y 292.756,Z 386.438,A -85,B 0,C 180,E1 -17225.515,E2 -17225.515} C_VEL
LIN {X 0,Y 287.35,Z 375.113,A -85,B 0,C 180,E1 -17226.876,E2 -17226.876} C_VEL
LIN {X 0,Y 285.543,Z 371.708,A -85,B 0,C 180,E1 -17227.279,E2 -17227.279} C_VEL
LIN {X 0,Y 284.289,Z 369.019,A -85,B 0,C 180,E1 -17227.574,E2 -17227.574} C_VEL
LIN {X 0,Y 284.099,Z 368.133,A -85,B 0,C 180,E1 -17227.663,E2 -17227.663} C_VEL
LIN {X 0,Y 284.203,Z 366.701,A -85,B 0,C 180,E1 -17230.011,E2 -17230.011} C_VEL
LIN {X 0,Y 284.176,Z 365.707,A -85,B 0,C 180,E1 -17232.103,E2 -17232.103} C_VEL
LIN {X 0,Y 284.254,Z 365.703,A -85,B 0,C 180,E1 -17236.189,E2 -17236.189} C_VEL
LIN {X 0,Y 284.305,Z 365.697,A -85,B 0,C 180,E1 -17240.023,E2 -17240.023} C_VEL
LIN {X 0,Y 284.348,Z 365.69,A -85,B 0,C 180,E1 -17243.616,E2 -17243.616} C_VEL
LIN {X 0,Y 284.306,Z 365.678,A -85,B 0,C 180,E1 -17247.189,E2 -17247.189} C_VEL
LIN {X 0,Y 284.357,Z 365.688,A -85,B 0,C 180,E1 -17250.376,E2 -17250.376} C_VEL
LIN {X 0,Y 284.376,Z 365.667,A -85,B 0,C 180,E1 -17253.586,E2 -17253.586} C_VEL
LIN {X 0,Y 284.365,Z 365.687,A -85,B 0,C 180,E1 -17256.707,E2 -17256.707} C_VEL
LIN {X 0,Y 284.401,Z 365.671,A -85,B 0,C 180,E1 -17261.261,E2 -17261.261} C_VEL
LIN {X 0,Y 284.49,Z 365.667,A -85,B 0,C 180,E1 -17264.459,E2 -17264.459} C_VEL
LIN {X 0,Y 284.488,Z 365.657,A -85,B 0,C 180,E1 -17268.601,E2 -17268.601} C_VEL
LIN {X 0,Y 284.657,Z 365.651,A -85,B 0,C 180,E1 -17271.481,E2 -17271.481} C_VEL
LIN {X 0,Y 284.6,Z 365.659,A -85,B 0,C 180,E1 -17274.331,E2 -17274.331} C_VEL
LIN {X 0,Y 284.839,Z 365.629,A -85,B 0,C 180,E1 -17278.476,E2 -17278.476} C_VEL
LIN {X 0,Y 284.238,Z 365.709,A -85,B 0,C 180,E1 -17279.656,E2 -17279.656} C_VEL
LIN {X 0,Y 282.595,Z 365.917,A -85,B 0,C 180,E1 -17280.811,E2 -17280.811} C_VEL
LIN {X 0,Y 278.641,Z 366.406,A -85,B 0,C 180,E1 -17283.13,E2 -17283.13} C_VEL
LIN {X 0,Y 277.548,Z 366.539,A -85,B 0,C 180,E1 -17284.343,E2 -17284.343} C_VEL
LIN {X 0,Y 277.476,Z 366.546,A -85,B 0,C 180,E1 -17284.754,E2 -17284.754} C_VEL
LIN {X 0,Y 277.651,Z 366.526,A -85,B 0,C 180,E1 -17287.271,E2 -17287.271} C_VEL
LIN {X 0,Y 277.504,Z 366.542,A -85,B 0,C 180,E1 -17290.211,E2 -17290.211} C_VEL
LIN {X 0,Y 277.432,Z 366.551,A -85,B 0,C 180,E1 -17294.674,E2 -17294.674} C_VEL
LIN {X 0,Y 277.342,Z 366.564,A -85,B 0,C 180,E1 -17299.234,E2 -17299.234} C_VEL
LIN {X 0,Y 277.317,Z 366.57,A -85,B 0,C 180,E1 -17304.171,E2 -17304.171} C_VEL
LIN {X 0,Y 277.323,Z 366.569,A -85,B 0,C 180,E1 -17307.506,E2 -17307.506} C_VEL
LIN {X 0,Y 277.336,Z 367.09,A -85,B 0,C 180,E1 -17308.782,E2 -17308.782} C_VEL
LIN {X 0,Y 277.759,Z 369.568,A -85,B 0,C 180,E1 -17312.097,E2 -17312.097} C_VEL
LIN {X 0,Y 278.306,Z 372.869,A -85,B 0,C 180,E1 -17316.092,E2 -17316.092} C_VEL
LIN {X 0,Y 278.759,Z 375.539,A -85,B 0,C 180,E1 -17319.072,E2 -17319.072} C_VEL
LIN {X 0,Y 279.319,Z 379.121,A -85,B 0,C 180,E1 -17322.793,E2 -17322.793} C_VEL
LIN {X 0,Y 279.686,Z 381.653,A -85,B 0,C 180,E1 -17325.285,E2 -17325.285} C_VEL
LIN {X 0,Y 279.844,Z 383.826,A -85,B 0,C 180,E1 -17327.307,E2 -17327.307} C_VEL
LIN {X 0,Y 279.384,Z 386.978,A -85,B 0,C 180,E1 -17330.1,E2 -17330.1} C_VEL
LIN {X 0,Y 279.09,Z 388.859,A -85,B 0,C 180,E1 -17331.581,E2 -17331.581} C_VEL
LIN {X 0,Y 280.106,Z 392.116,A -85,B 0,C 180,E1 -17331.858,E2 -17331.858} C_VEL
LIN {X 0,Y 284.936,Z 404.617,A -85,B 0,C 180,E1 -17333.137,E2 -17333.137} C_VEL
LIN {X 0,Y 289.094,Z 418.814,A -85,B 0,C 180,E1 -17334.602,E2 -17334.602} C_VEL
LIN {X 0,Y 292.123,Z 432.915,A -85,B 0,C 180,E1 -17336.134,E2 -17336.134} C_VEL
LIN {X 0,Y 293.902,Z 445.123,A -85,B 0,C 180,E1 -17337.553,E2 -17337.553} C_VEL
LIN {X 0,Y 294.945,Z 458.471,A -85,B 0,C 180,E1 -17339.255,E2 -17339.255} C_VEL
LIN {X 0,Y 292.087,Z 471.665,A -85,B 0,C 180,E1 -17340.841,E2 -17340.841} C_VEL
LIN {X 0,Y 288.989,Z 484.131,A -85,B 0,C 180,E1 -17342.676,E2 -17342.676} C_VEL
LIN {X 0,Y 285.785,Z 496.368,A -85,B 0,C 180,E1 -17344.9,E2 -17344.9} C_VEL
LIN {X 0,Y 283.005,Z 507.274,A -85,B 0,C 180,E1 -17347.362,E2 -17347.362} C_VEL
LIN {X 0,Y 280.494,Z 516.361,A -85,B 0,C 180,E1 -17349.848,E2 -17349.848} C_VEL
LIN {X 0,Y 278.673,Z 523.92,A -85,B 0,C 180,E1 -17352.385,E2 -17352.385} C_VEL
LIN {X 0,Y 277.074,Z 530.982,A -85,B 0,C 180,E1 -17355.307,E2 -17355.307} C_VEL
LIN {X 0,Y 275.992,Z 536.546,A -85,B 0,C 180,E1 -17358.246,E2 -17358.246} C_VEL
LIN {X 0,Y 275.472,Z 540.768,A -85,B 0,C 180,E1 -17361.195,E2 -17361.195} C_VEL
LIN {X 0,Y 275.347,Z 544.042,A -85,B 0,C 180,E1 -17364.527,E2 -17364.527} C_VEL
LIN {X 0,Y 275.373,Z 545.513,A -85,B 0,C 180,E1 -17367.075,E2 -17367.075} C_VEL
LIN {X 0,Y 275.41,Z 546.12,A -85,B 0,C 180,E1 -17370.001,E2 -17370.001} C_VEL
LIN {X 0,Y 275.377,Z 545.503,A -85,B 0,C 180,E1 -17372.926,E2 -17372.926} C_VEL
LIN {X 0,Y 275.389,Z 543.716,A -85,B 0,C 180,E1 -17375.86,E2 -17375.86} C_VEL
LIN {X 0,Y 275.473,Z 540.735,A -85,B 0,C 180,E1 -17378.806,E2 -17378.806} C_VEL
LIN {X 0,Y 275.994,Z 536.507,A -85,B 0,C 180,E1 -17381.755,E2 -17381.755} C_VEL
LIN {X 0,Y 277.076,Z 530.927,A -85,B 0,C 180,E1 -17384.694,E2 -17384.694} C_VEL
LIN {X 0,Y 278.674,Z 523.842,A -85,B 0,C 180,E1 -17387.616,E2 -17387.616} C_VEL
LIN {X 0,Y 280.815,Z 515.042,A -85,B 0,C 180,E1 -17390.511,E2 -17390.511} C_VEL
LIN {X 0,Y 283.351,Z 505.717,A -85,B 0,C 180,E1 -17392.996,E2 -17392.996} C_VEL
LIN {X 0,Y 285.81,Z 496.244,A -85,B 0,C 180,E1 -17395.099,E2 -17395.099} C_VEL
LIN {X 0,Y 288.974,Z 483.974,A -85,B 0,C 180,E1 -17397.326,E2 -17397.326} C_VEL
LIN {X 0,Y 292.111,Z 471.48,A -85,B 0,C 180,E1 -17399.157,E2 -17399.157} C_VEL
LIN {X 0,Y 294.905,Z 458.377,A -85,B 0,C 180,E1 -17400.732,E2 -17400.732} C_VEL
LIN {X 0,Y 293.879,Z 445.034,A -85,B 0,C 180,E1 -17402.428,E2 -17402.428} C_VEL
LIN {X 0,Y 291.82,Z 431.318,A -85,B 0,C 180,E1 -17404.017,E2 -17404.017} C_VEL
LIN {X 0,Y 288.775,Z 417.753,A -85,B 0,C 180,E1 -17405.482,E2 -17405.482} C_VEL
LIN {X 0,Y 284.593,Z 403.752,A -85,B 0,C 180,E1 -17406.918,E2 -17406.918} C_VEL
LIN {X 0,Y 280.157,Z 392.287,A -85,B 0,C 180,E1 -17408.088,E2 -17408.088} C_VEL
LIN {X 0,Y 279.103,Z 389.078,A -85,B 0,C 180,E1 -17408.369,E2 -17408.369} C_VEL
LIN {X 0,Y 279.055,Z 388.647,A -85,B 0,C 180,E1 -17408.426,E2 -17408.426} C_VEL
LIN {X 0,Y 279.631,Z 385.607,A -85,B 0,C 180,E1 -17411.063,E2 -17411.063} C_VEL
LIN {X 0,Y 279.862,Z 383.164,A -85,B 0,C 180,E1 -17413.26,E2 -17413.26} C_VEL
LIN {X 0,Y 279.366,Z 379.384,A -85,B 0,C 180,E1 -17416.85,E2 -17416.85} C_VEL
LIN {X 0,Y 279.035,Z 377.195,A -85,B 0,C 180,E1 -17419.091,E2 -17419.091} C_VEL
LIN {X 0,Y 278.484,Z 373.838,A -85,B 0,C 180,E1 -17422.722,E2 -17422.722} C_VEL
LIN {X 0,Y 277.917,Z 370.578,A -85,B 0,C 180,E1 -17426.566,E2 -17426.566} C_VEL
LIN {X 0,Y 277.569,Z 368.24,A -85,B 0,C 180,E1 -17429.576,E2 -17429.576} C_VEL
LIN {X 0,Y 277.333,Z 367.038,A -85,B 0,C 180,E1 -17431.218,E2 -17431.218} C_VEL
LIN {X 0,Y 277.36,Z 366.562,A -85,B 0,C 180,E1 -17432.864,E2 -17432.864} C_VEL
LIN {X 0,Y 277.332,Z 366.565,A -85,B 0,C 180,E1 -17436.08,E2 -17436.08} C_VEL
LIN {X 0,Y 277.348,Z 366.562,A -85,B 0,C 180,E1 -17440.767,E2 -17440.767} C_VEL
LIN {X 0,Y 277.438,Z 366.556,A -85,B 0,C 180,E1 -17445.326,E2 -17445.326} C_VEL
LIN {X 0,Y 277.51,Z 366.546,A -85,B 0,C 180,E1 -17449.789,E2 -17449.789} C_VEL
LIN {X 0,Y 277.657,Z 366.526,A -85,B 0,C 180,E1 -17452.729,E2 -17452.729} C_VEL
LIN {X 0,Y 277.824,Z 366.503,A -85,B 0,C 180,E1 -17458.551,E2 -17458.551} C_VEL
LIN {X 0,Y 277.825,Z 366.505,A -85,B 0,C 180,E1 -17461.45,E2 -17461.45} C_VEL
LIN {X 0,Y 277.657,Z 366.519,A -85,B 0,C 180,E1 -17467.271,E2 -17467.271} C_VEL
LIN {X 0,Y 277.51,Z 366.535,A -85,B 0,C 180,E1 -17470.211,E2 -17470.211} C_VEL
LIN {X 0,Y 277.438,Z 366.535,A -85,B 0,C 180,E1 -17474.674,E2 -17474.674} C_VEL
LIN {X 0,Y 277.346,Z 366.539,A -85,B 0,C 180,E1 -17479.234,E2 -17479.234} C_VEL
LIN {X 0,Y 277.296,Z 366.569,A -85,B 0,C 180,E1 -17484.158,E2 -17484.158} C_VEL
LIN {X 0,Y 277.327,Z 366.541,A -85,B 0,C 180,E1 -17487.504,E2 -17487.504} C_VEL
LIN {X 0,Y 277.275,Z 366.573,A -85,B 0,C 180,E1 -17490.481,E2 -17490.481} C_VEL
LIN {X 0,Y 277.257,Z 366.555,A -85,B 0,C 180,E1 -17493.895,E2 -17493.895} C_VEL
LIN {X 0,Y 277.284,Z 366.572,A -85,B 0,C 180,E1 -17497.467,E2 -17497.467} C_VEL
LIN {X 0,Y 277.212,Z 366.58,A -85,B 0,C 180,E1 -17501.236,E2 -17501.236} C_VEL
LIN {X 0,Y 277.172,Z 366.591,A -85,B 0,C 180,E1 -17505.233,E2 -17505.233} C_VEL
LIN {X 0,Y 277.135,Z 366.595,A -85,B 0,C 180,E1 -17507.343,E2 -17507.343} C_VEL
LIN {X 0,Y 277.146,Z 367.495,A -85,B 0,C 180,E1 -17509.531,E2 -17509.531} C_VEL
LIN {X 0,Y 277.103,Z 368.667,A -85,B 0,C 180,E1 -17511.379,E2 -17511.379} C_VEL
LIN {X 0,Y 278.207,Z 371.636,A -85,B 0,C 180,E1 -17511.675,E2 -17511.675} C_VEL
LIN {X 0,Y 279.505,Z 373.677,A -85,B 0,C 180,E1 -17511.966,E2 -17511.966} C_VEL
LIN {X 0,Y 285.534,Z 385.971,A -85,B 0,C 180,E1 -17513.518,E2 -17513.518} C_VEL
LIN {X 0,Y 290.375,Z 397.589,A -85,B 0,C 180,E1 -17514.997,E2 -17514.997} C_VEL
LIN {X 0,Y 294.704,Z 411.029,A -85,B 0,C 180,E1 -17516.735,E2 -17516.735} C_VEL
LIN {X 0,Y 297.712,Z 423.573,A -85,B 0,C 180,E1 -17518.436,E2 -17518.436} C_VEL
LIN {X 0,Y 298.055,Z 427.033,A -85,B 0,C 180,E1 -17518.876,E2 -17518.876} C_VEL
LIN {X 0,Y 295.258,Z 440.933,A -85,B 0,C 180,E1 -17520.401,E2 -17520.401} C_VEL
LIN {X 0,Y 292.512,Z 453.124,A -85,B 0,C 180,E1 -17522.061,E2 -17522.061} C_VEL
LIN {X 0,Y 289.491,Z 465.259,A -85,B 0,C 180,E1 -17524.088,E2 -17524.088} C_VEL
LIN {X 0,Y 286.82,Z 475.398,A -85,B 0,C 180,E1 -17526.152,E2 -17526.152} C_VEL
LIN {X 0,Y 284.05,Z 485.312,A -85,B 0,C 180,E1 -17528.595,E2 -17528.595} C_VEL
LIN {X 0,Y 281.708,Z 493.525,A -85,B 0,C 180,E1 -17531.075,E2 -17531.075} C_VEL
LIN {X 0,Y 280.084,Z 499.444,A -85,B 0,C 180,E1 -17533.227,E2 -17533.227} C_VEL
LIN {X 0,Y 278.289,Z 505.953,A -85,B 0,C 180,E1 -17536.118,E2 -17536.118} C_VEL
LIN {X 0,Y 277.073,Z 511.028,A -85,B 0,C 180,E1 -17539.033,E2 -17539.033} C_VEL
LIN {X 0,Y 276.376,Z 513.951,A -85,B 0,C 180,E1 -17541.223,E2 -17541.223} C_VEL
LIN {X 0,Y 275.857,Z 516.805,A -85,B 0,C 180,E1 -17544.15,E2 -17544.15} C_VEL
LIN {X 0,Y 275.553,Z 518.52,A -85,B 0,C 180,E1 -17547.075,E2 -17547.075} C_VEL
LIN {X 0,Y 275.455,Z 519.119,A -85,B 0,C 180,E1 -17549.999,E2 -17549.999} C_VEL
LIN {X 0,Y 275.552,Z 518.56,A -85,B 0,C 180,E1 -17552.923,E2 -17552.923} C_VEL
LIN {X 0,Y 275.858,Z 516.897,A -85,B 0,C 180,E1 -17555.848,E2 -17555.848} C_VEL
LIN {X 0,Y 276.37,Z 514.092,A -85,B 0,C 180,E1 -17558.776,E2 -17558.776} C_VEL
LIN {X 0,Y 277.289,Z 510.069,A -85,B 0,C 180,E1 -17561.698,E2 -17561.698} C_VEL
LIN {X 0,Y 278.611,Z 504.728,A -85,B 0,C 180,E1 -17564.61,E2 -17564.61} C_VEL
LIN {X 0,Y 280.047,Z 499.73,A -85,B 0,C 180,E1 -17566.774,E2 -17566.774} C_VEL
LIN {X 0,Y 281.907,Z 492.778,A -85,B 0,C 180,E1 -17569.288,E2 -17569.288} C_VEL
LIN {X 0,Y 284.35,Z 484.393,A -85,B 0,C 180,E1 -17571.761,E2 -17571.761} C_VEL
LIN {X 0,Y 287.134,Z 474.291,A -85,B 0,C 180,E1 -17574.203,E2 -17574.203} C_VEL
LIN {X 0,Y 289.964,Z 463.537,A -85,B 0,C 180,E1 -17576.334,E2 -17576.334} C_VEL
LIN {X 0,Y 292.655,Z 452.68,A -85,B 0,C 180,E1 -17578.117,E2 -17578.117} C_VEL
LIN {X 0,Y 295.413,Z 440.427,A -85,B 0,C 180,E1 -17579.776,E2 -17579.776} C_VEL
LIN {X 0,Y 298.121,Z 427.015,A -85,B 0,C 180,E1 -17581.24,E2 -17581.24} C_VEL
LIN {X 0,Y 297.94,Z 424.541,A -85,B 0,C 180,E1 -17581.547,E2 -17581.547} C_VEL
LIN {X 0,Y 295.086,Z 412.362,A -85,B 0,C 180,E1 -17583.215,E2 -17583.215} C_VEL
LIN {X 0,Y 291.158,Z 399.802,A -85,B 0,C 180,E1 -17584.845,E2 -17584.845} C_VEL
LIN {X 0,Y 286.137,Z 387.13,A -85,B 0,C 180,E1 -17586.448,E2 -17586.448} C_VEL
LIN {X 0,Y 280.586,Z 375.828,A -85,B 0,C 180,E1 -17587.908,E2 -17587.908} C_VEL
LIN {X 0,Y 278.631,Z 372.219,A -85,B 0,C 180,E1 -17588.365,E2 -17588.365} C_VEL
LIN {X 0,Y 277.27,Z 369.371,A -85,B 0,C 180,E1 -17588.701,E2 -17588.701} C_VEL
LIN {X 0,Y 277.129,Z 368.514,A -85,B 0,C 180,E1 -17588.828,E2 -17588.828} C_VEL
LIN {X 0,Y 277.155,Z 367.113,A -85,B 0,C 180,E1 -17591.245,E2 -17591.245} C_VEL
LIN {X 0,Y 277.142,Z 366.584,A -85,B 0,C 180,E1 -17593.21,E2 -17593.21} C_VEL
LIN {X 0,Y 277.213,Z 366.581,A -85,B 0,C 180,E1 -17597.325,E2 -17597.325} C_VEL
LIN {X 0,Y 277.273,Z 366.572,A -85,B 0,C 180,E1 -17601.789,E2 -17601.789} C_VEL
LIN {X 0,Y 277.302,Z 366.569,A -85,B 0,C 180,E1 -17604.344,E2 -17604.344} C_VEL
LIN {X 0,Y 277.243,Z 366.561,A -85,B 0,C 180,E1 -17607.836,E2 -17607.836} C_VEL
LIN {X 0,Y 277.288,Z 366.561,A -85,B 0,C 180,E1 -17611.212,E2 -17611.212} C_VEL
LIN {X 0,Y 277.312,Z 366.556,A -85,B 0,C 180,E1 -17614.479,E2 -17614.479} C_VEL
LIN {X 0,Y 277.283,Z 366.561,A -85,B 0,C 180,E1 -17617.654,E2 -17617.654} C_VEL
LIN {X 0,Y 277.343,Z 366.542,A -85,B 0,C 180,E1 -17620.766,E2 -17620.766} C_VEL
LIN {X 0,Y 277.433,Z 366.534,A -85,B 0,C 180,E1 -17625.326,E2 -17625.326} C_VEL
LIN {X 0,Y 277.505,Z 366.54,A -85,B 0,C 180,E1 -17629.788,E2 -17629.788} C_VEL
LIN {X 0,Y 277.651,Z 366.526,A -85,B 0,C 180,E1 -17632.729,E2 -17632.729} C_VEL
LIN {X 0,Y 277.82,Z 366.504,A -85,B 0,C 180,E1 -17638.55,E2 -17638.55} C_VEL
LIN {X 0,Y 277.82,Z 366.506,A -85,B 0,C 180,E1 -17641.449,E2 -17641.449} C_VEL
LIN {X 0,Y 277.476,Z 366.546,A -85,B 0,C 180,E1 -17644.754,E2 -17644.754} C_VEL
LIN {X 0,Y 276.852,Z 366.626,A -85,B 0,C 180,E1 -17645.968,E2 -17645.968} C_VEL
LIN {X 0,Y 274.008,Z 366.979,A -85,B 0,C 180,E1 -17647.945,E2 -17647.945} C_VEL
LIN {X 0,Y 271.557,Z 367.284,A -85,B 0,C 180,E1 -17649.552,E2 -17649.552} C_VEL
LIN {X 0,Y 270.488,Z 367.419,A -85,B 0,C 180,E1 -17650.798,E2 -17650.798} C_VEL
LIN {X 0,Y 270.395,Z 367.423,A -85,B 0,C 180,E1 -17651.22,E2 -17651.22} C_VEL
LIN {X 0,Y 270.378,Z 367.425,A -85,B 0,C 180,E1 -17655.901,E2 -17655.901} C_VEL
LIN {X 0,Y 270.29,Z 367.439,A -85,B 0,C 180,E1 -17660.602,E2 -17660.602} C_VEL
LIN {X 0,Y 270.272,Z 367.447,A -85,B 0,C 180,E1 -17664.586,E2 -17664.586} C_VEL
LIN {X 0,Y 270.261,Z 367.449,A -85,B 0,C 180,E1 -17666.236,E2 -17666.236} C_VEL
LIN {X 0,Y 270.317,Z 367.91,A -85,B 0,C 180,E1 -17667.903,E2 -17667.903} C_VEL
LIN {X 0,Y 270.711,Z 370.352,A -85,B 0,C 180,E1 -17671.28,E2 -17671.28} C_VEL
LIN {X 0,Y 271.129,Z 373.097,A -85,B 0,C 180,E1 -17674.769,E2 -17674.769} C_VEL
LIN {X 0,Y 271.778,Z 376.855,A -85,B 0,C 180,E1 -17679.125,E2 -17679.125} C_VEL
LIN {X 0,Y 272.213,Z 379.684,A -85,B 0,C 180,E1 -17682.165,E2 -17682.165} C_VEL
LIN {X 0,Y 272.746,Z 383.67,A -85,B 0,C 180,E1 -17686.177,E2 -17686.177} C_VEL
LIN {X 0,Y 272.656,Z 385.996,A -85,B 0,C 180,E1 -17688.375,E2 -17688.375} C_VEL
LIN {X 0,Y 272.243,Z 388.296,A -85,B 0,C 180,E1 -17690.423,E2 -17690.423} C_VEL
LIN {X 0,Y 273.182,Z 391.529,A -85,B 0,C 180,E1 -17690.701,E2 -17690.701} C_VEL
LIN {X 0,Y 274.466,Z 394.442,A -85,B 0,C 180,E1 -17691.031,E2 -17691.031} C_VEL
LIN {X 0,Y 279.523,Z 408.153,A -85,B 0,C 180,E1 -17692.52,E2 -17692.52} C_VEL
LIN {X 0,Y 283.256,Z 421.318,A -85,B 0,C 180,E1 -17693.963,E2 -17693.963} C_VEL
LIN {X 0,Y 285.869,Z 434.235,A -85,B 0,C 180,E1 -17695.446,E2 -17695.446} C_VEL
LIN {X 0,Y 287.546,Z 446.16,A -85,B 0,C 180,E1 -17696.908,E2 -17696.908} C_VEL
LIN {X 0,Y 288.461,Z 458.287,A -85,B 0,C 180,E1 -17698.51,E2 -17698.51} C_VEL
LIN {X 0,Y 288.176,Z 461.574,A -85,B 0,C 180,E1 -17698.938,E2 -17698.938} C_VEL
LIN {X 0,Y 284.912,Z 474.891,A -85,B 0,C 180,E1 -17700.643,E2 -17700.643} C_VEL
LIN {X 0,Y 281.794,Z 486.766,A -85,B 0,C 180,E1 -17702.524,E2 -17702.524} C_VEL
LIN {X 0,Y 278.865,Z 497.664,A -85,B 0,C 180,E1 -17704.632,E2 -17704.632} C_VEL
LIN {X 0,Y 276.351,Z 506.922,A -85,B 0,C 180,E1 -17706.785,E2 -17706.785} C_VEL
LIN {X 0,Y 273.769,Z 516.011,A -85,B 0,C 180,E1 -17709.331,E2 -17709.331} C_VEL
LIN {X 0,Y 271.816,Z 523.569,A -85,B 0,C 180,E1 -17711.925,E2 -17711.925} C_VEL
LIN {X 0,Y 270.119,Z 530.631,A -85,B 0,C 180,E1 -17714.92,E2 -17714.92} C_VEL
LIN {X 0,Y 268.991,Z 536.197,A -85,B 0,C 180,E1 -17717.936,E2 -17717.936} C_VEL
LIN {X 0,Y 268.409,Z 540.418,A -85,B 0,C 180,E1 -17720.962,E2 -17720.962} C_VEL
LIN {X 0,Y 268.239,Z 543.389,A -85,B 0,C 180,E1 -17723.985,E2 -17723.985} C_VEL
LIN {X 0,Y 268.278,Z 545.165,A -85,B 0,C 180,E1 -17726.997,E2 -17726.997} C_VEL
LIN {X 0,Y 268.328,Z 545.773,A -85,B 0,C 180,E1 -17730.001,E2 -17730.001} C_VEL
LIN {X 0,Y 268.283,Z 545.154,A -85,B 0,C 180,E1 -17733.004,E2 -17733.004} C_VEL
LIN {X 0,Y 268.298,Z 543.367,A -85,B 0,C 180,E1 -17736.015,E2 -17736.015} C_VEL
LIN {X 0,Y 268.41,Z 540.384,A -85,B 0,C 180,E1 -17739.039,E2 -17739.039} C_VEL
LIN {X 0,Y 268.993,Z 536.156,A -85,B 0,C 180,E1 -17742.065,E2 -17742.065} C_VEL
LIN {X 0,Y 270.124,Z 530.573,A -85,B 0,C 180,E1 -17745.081,E2 -17745.081} C_VEL
LIN {X 0,Y 271.818,Z 523.488,A -85,B 0,C 180,E1 -17748.076,E2 -17748.076} C_VEL
LIN {X 0,Y 274.117,Z 514.689,A -85,B 0,C 180,E1 -17751.036,E2 -17751.036} C_VEL
LIN {X 0,Y 276.771,Z 505.364,A -85,B 0,C 180,E1 -17753.575,E2 -17753.575} C_VEL
LIN {X 0,Y 279.322,Z 495.89,A -85,B 0,C 180,E1 -17755.724,E2 -17755.724} C_VEL
LIN {X 0,Y 282.656,Z 483.621,A -85,B 0,C 180,E1 -17757.99,E2 -17757.99} C_VEL
LIN {X 0,Y 285.911,Z 471.127,A -85,B 0,C 180,E1 -17759.853,E2 -17759.853} C_VEL
LIN {X 0,Y 288.443,Z 459.915,A -85,B 0,C 180,E1 -17761.234,E2 -17761.234} C_VEL
LIN {X 0,Y 287.523,Z 446.046,A -85,B 0,C 180,E1 -17763.074,E2 -17763.074} C_VEL
LIN {X 0,Y 285.838,Z 434.009,A -85,B 0,C 180,E1 -17764.545,E2 -17764.545} C_VEL
LIN {X 0,Y 282.874,Z 419.984,A -85,B 0,C 180,E1 -17766.153,E2 -17766.153} C_VEL
LIN {X 0,Y 278.846,Z 406.145,A -85,B 0,C 180,E1 -17767.669,E2 -17767.669} C_VEL
LIN {X 0,Y 273.633,Z 392.42,A -85,B 0,C 180,E1 -17769.144,E2 -17769.144} C_VEL
LIN {X 0,Y 272.384,Z 389.325,A -85,B 0,C 180,E1 -17769.473,E2 -17769.473} C_VEL
LIN {X 0,Y 272.227,Z 388.266,A -85,B 0,C 180,E1 -17769.568,E2 -17769.568} C_VEL
LIN {X 0,Y 272.707,Z 385.467,A -85,B 0,C 180,E1 -17772.072,E2 -17772.072} C_VEL
LIN {X 0,Y 272.772,Z 383.355,A -85,B 0,C 180,E1 -17774.08,E2 -17774.08} C_VEL
LIN {X 0,Y 272.208,Z 379.595,A -85,B 0,C 180,E1 -17777.834,E2 -17777.834} C_VEL
LIN {X 0,Y 271.656,Z 376.074,A -85,B 0,C 180,E1 -17781.618,E2 -17781.618} C_VEL
LIN {X 0,Y 271.013,Z 372.348,A -85,B 0,C 180,E1 -17786.083,E2 -17786.083} C_VEL
LIN {X 0,Y 270.471,Z 369.053,A -85,B 0,C 180,E1 -17790.416,E2 -17790.416} C_VEL
LIN {X 0,Y 270.331,Z 367.838,A -85,B 0,C 180,E1 -17792.12,E2 -17792.12} C_VEL
LIN {X 0,Y 270.266,Z 367.446,A -85,B 0,C 180,E1 -17793.764,E2 -17793.764} C_VEL
LIN {X 0,Y 270.236,Z 367.45,A -85,B 0,C 180,E1 -17797.039,E2 -17797.039} C_VEL
LIN {X 0,Y 270.305,Z 367.441,A -85,B 0,C 180,E1 -17800.245,E2 -17800.245} C_VEL
LIN {X 0,Y 270.406,Z 367.432,A -85,B 0,C 180,E1 -17804.936,E2 -17804.936} C_VEL
LIN {X 0,Y 270.445,Z 367.427,A -85,B 0,C 180,E1 -17809.519,E2 -17809.519} C_VEL
LIN {X 0,Y 270.615,Z 367.404,A -85,B 0,C 180,E1 -17812.539,E2 -17812.539} C_VEL
LIN {X 0,Y 270.79,Z 367.38,A -85,B 0,C 180,E1 -17818.513,E2 -17818.513} C_VEL
LIN {X 0,Y 270.791,Z 367.381,A -85,B 0,C 180,E1 -17821.487,E2 -17821.487} C_VEL
LIN {X 0,Y 270.615,Z 367.396,A -85,B 0,C 180,E1 -17827.461,E2 -17827.461} C_VEL
LIN {X 0,Y 270.445,Z 367.413,A -85,B 0,C 180,E1 -17830.481,E2 -17830.481} C_VEL
LIN {X 0,Y 270.406,Z 367.416,A -85,B 0,C 180,E1 -17835.065,E2 -17835.065} C_VEL
LIN {X 0,Y 270.303,Z 367.41,A -85,B 0,C 180,E1 -17839.756,E2 -17839.756} C_VEL
LIN {X 0,Y 270.241,Z 367.445,A -85,B 0,C 180,E1 -17844.589,E2 -17844.589} C_VEL
LIN {X 0,Y 270.273,Z 367.421,A -85,B 0,C 180,E1 -17847.909,E2 -17847.909} C_VEL
LIN {X 0,Y 270.187,Z 367.451,A -85,B 0,C 180,E1 -17851.348,E2 -17851.348} C_VEL
LIN {X 0,Y 270.218,Z 367.442,A -85,B 0,C 180,E1 -17854.903,E2 -17854.903} C_VEL
LIN {X 0,Y 270.225,Z 367.451,A -85,B 0,C 180,E1 -17858.717,E2 -17858.717} C_VEL
LIN {X 0,Y 270.168,Z 367.459,A -85,B 0,C 180,E1 -17863.249,E2 -17863.249} C_VEL
LIN {X 0,Y 270.099,Z 367.472,A -85,B 0,C 180,E1 -17867.427,E2 -17867.427} C_VEL
LIN {X 0,Y 270.117,Z 368.995,A -85,B 0,C 180,E1 -17870.165,E2 -17870.165} C_VEL
LIN {X 0,Y 271.255,Z 372.073,A -85,B 0,C 180,E1 -17870.504,E2 -17870.504} C_VEL
LIN {X 0,Y 272.717,Z 374.405,A -85,B 0,C 180,E1 -17870.853,E2 -17870.853} C_VEL
LIN {X 0,Y 278.802,Z 386.471,A -85,B 0,C 180,E1 -17872.492,E2 -17872.492} C_VEL
LIN {X 0,Y 283.658,Z 397.898,A -85,B 0,C 180,E1 -17874.034,E2 -17874.034} C_VEL
LIN {X 0,Y 287.581,Z 409.682,A -85,B 0,C 180,E1 -17875.63,E2 -17875.63} C_VEL
LIN {X 0,Y 290.335,Z 420.11,A -85,B 0,C 180,E1 -17877.079,E2 -17877.079} C_VEL
LIN {X 0,Y 291.821,Z 427.458,A -85,B 0,C 180,E1 -17878.141,E2 -17878.141} C_VEL
LIN {X 0,Y 289.391,Z 439.923,A -85,B 0,C 180,E1 -17879.538,E2 -17879.538} C_VEL
LIN {X 0,Y 286.55,Z 452.318,A -85,B 0,C 180,E1 -17881.227,E2 -17881.227} C_VEL
LIN {X 0,Y 283.388,Z 464.373,A -85,B 0,C 180,E1 -17883.227,E2 -17883.227} C_VEL
LIN {X 0,Y 280.769,Z 474.138,A -85,B 0,C 180,E1 -17885.211,E2 -17885.211} C_VEL
LIN {X 0,Y 277.816,Z 484.325,A -85,B 0,C 180,E1 -17887.699,E2 -17887.699} C_VEL
LIN {X 0,Y 275.287,Z 492.776,A -85,B 0,C 180,E1 -17890.228,E2 -17890.228} C_VEL
LIN {X 0,Y 273.259,Z 499.796,A -85,B 0,C 180,E1 -17892.796,E2 -17892.796} C_VEL
LIN {X 0,Y 271.369,Z 506.304,A -85,B 0,C 180,E1 -17895.756,E2 -17895.756} C_VEL
LIN {X 0,Y 270.092,Z 511.378,A -85,B 0,C 180,E1 -17898.746,E2 -17898.746} C_VEL
LIN {X 0,Y 269.344,Z 514.301,A -85,B 0,C 180,E1 -17900.992,E2 -17900.992} C_VEL
LIN {X 0,Y 268.789,Z 517.154,A -85,B 0,C 180,E1 -17903.996,E2 -17903.996} C_VEL
LIN {X 0,Y 268.484,Z 518.868,A -85,B 0,C 180,E1 -17906.998,E2 -17906.998} C_VEL
LIN {X 0,Y 268.372,Z 519.466,A -85,B 0,C 180,E1 -17909.999,E2 -17909.999} C_VEL
LIN {X 0,Y 268.483,Z 518.907,A -85,B 0,C 180,E1 -17913,E2 -17913} C_VEL
LIN {X 0,Y 268.79,Z 517.245,A -85,B 0,C 180,E1 -17916.003,E2 -17916.003} C_VEL
LIN {X 0,Y 269.337,Z 514.44,A -85,B 0,C 180,E1 -17919.007,E2 -17919.007} C_VEL
LIN {X 0,Y 270.336,Z 510.416,A -85,B 0,C 180,E1 -17922.003,E2 -17922.003} C_VEL
LIN {X 0,Y 271.739,Z 505.075,A -85,B 0,C 180,E1 -17924.988,E2 -17924.988} C_VEL
LIN {X 0,Y 273.219,Z 500.079,A -85,B 0,C 180,E1 -17927.206,E2 -17927.206} C_VEL
LIN {X 0,Y 275.192,Z 493.125,A -85,B 0,C 180,E1 -17929.778,E2 -17929.778} C_VEL
LIN {X 0,Y 277.768,Z 484.739,A -85,B 0,C 180,E1 -17932.304,E2 -17932.304} C_VEL
LIN {X 0,Y 280.666,Z 474.636,A -85,B 0,C 180,E1 -17934.798,E2 -17934.798} C_VEL
LIN {X 0,Y 283.722,Z 463.422,A -85,B 0,C 180,E1 -17937.054,E2 -17937.054} C_VEL
LIN {X 0,Y 286.728,Z 451.857,A -85,B 0,C 180,E1 -17938.952,E2 -17938.952} C_VEL
LIN {X 0,Y 289.571,Z 439.366,A -85,B 0,C 180,E1 -17940.642,E2 -17940.642} C_VEL
LIN {X 0,Y 291.755,Z 428.9,A -85,B 0,C 180,E1 -17941.803,E2 -17941.803} C_VEL
LIN {X 0,Y 291.633,Z 426.151,A -85,B 0,C 180,E1 -17942.164,E2 -17942.164} C_VEL
LIN {X 0,Y 288.841,Z 414.001,A -85,B 0,C 180,E1 -17943.9,E2 -17943.9} C_VEL
LIN {X 0,Y 285.076,Z 401.877,A -85,B 0,C 180,E1 -17945.555,E2 -17945.555} C_VEL
LIN {X 0,Y 280.217,Z 389.508,A -85,B 0,C 180,E1 -17947.221,E2 -17947.221} C_VEL
LIN {X 0,Y 274.268,Z 377.195,A -85,B 0,C 180,E1 -17948.897,E2 -17948.897} C_VEL
LIN {X 0,Y 271.929,Z 372.967,A -85,B 0,C 180,E1 -17949.477,E2 -17949.477} C_VEL
LIN {X 0,Y 270.445,Z 370.3,A -85,B 0,C 180,E1 -17949.848,E2 -17949.848} C_VEL
LIN {X 0,Y 270.139,Z 368.974,A -85,B 0,C 180,E1 -17949.96,E2 -17949.96} C_VEL
LIN {X 0,Y 270.096,Z 367.533,A -85,B 0,C 180,E1 -17952.572,E2 -17952.572} C_VEL
LIN {X 0,Y 270.164,Z 367.458,A -85,B 0,C 180,E1 -17956.75,E2 -17956.75} C_VEL
LIN {X 0,Y 270.221,Z 367.449,A -85,B 0,C 180,E1 -17961.282,E2 -17961.282} C_VEL
LIN {X 0,Y 270.213,Z 367.447,A -85,B 0,C 180,E1 -17965.096,E2 -17965.096} C_VEL
LIN {X 0,Y 270.199,Z 367.452,A -85,B 0,C 180,E1 -17969.13,E2 -17969.13} C_VEL
LIN {X 0,Y 270.263,Z 367.424,A -85,B 0,C 180,E1 -17972.145,E2 -17972.145} C_VEL
LIN {X 0,Y 270.275,Z 367.441,A -85,B 0,C 180,E1 -17975.519,E2 -17975.519} C_VEL
LIN {X 0,Y 270.3,Z 367.414,A -85,B 0,C 180,E1 -17980.244,E2 -17980.244} C_VEL
LIN {X 0,Y 270.401,Z 367.415,A -85,B 0,C 180,E1 -17984.935,E2 -17984.935} C_VEL
LIN {X 0,Y 270.44,Z 367.418,A -85,B 0,C 180,E1 -17989.519,E2 -17989.519} C_VEL
LIN {X 0,Y 270.609,Z 367.402,A -85,B 0,C 180,E1 -17992.539,E2 -17992.539} C_VEL
LIN {X 0,Y 270.786,Z 367.38,A -85,B 0,C 180,E1 -17998.513,E2 -17998.513} C_VEL
LIN {X 0,Y 270.786,Z 367.383,A -85,B 0,C 180,E1 -18001.487,E2 -18001.487} C_VEL
LIN {X 0,Y 270.609,Z 367.404,A -85,B 0,C 180,E1 -18007.461,E2 -18007.461} C_VEL
LIN {X 0,Y 270.439,Z 367.423,A -85,B 0,C 180,E1 -18010.481,E2 -18010.481} C_VEL
LIN {X 0,Y 270.395,Z 367.423,A -85,B 0,C 180,E1 -18011.22,E2 -18011.22} C_VEL
LIN {X 0,Y 269.701,Z 367.51,A -85,B 0,C 180,E1 -18012.465,E2 -18012.465} C_VEL
LIN {X 0,Y 266.814,Z 367.874,A -85,B 0,C 180,E1 -18014.491,E2 -18014.491} C_VEL
LIN {X 0,Y 264.371,Z 368.178,A -85,B 0,C 180,E1 -18016.139,E2 -18016.139} C_VEL
LIN {X 0,Y 263.32,Z 368.309,A -85,B 0,C 180,E1 -18017.417,E2 -18017.417} C_VEL
LIN {X 0,Y 263.232,Z 368.316,A -85,B 0,C 180,E1 -18017.85,E2 -18017.85} C_VEL
LIN {X 0,Y 263.215,Z 368.32,A -85,B 0,C 180,E1 -18020.851,E2 -18020.851} C_VEL
LIN {X 0,Y 263.206,Z 368.327,A -85,B 0,C 180,E1 -18025.291,E2 -18025.291} C_VEL
LIN {X 0,Y 263.281,Z 368.771,A -85,B 0,C 180,E1 -18026.987,E2 -18026.987} C_VEL
LIN {X 0,Y 263.784,Z 371.91,A -85,B 0,C 180,E1 -18031.508,E2 -18031.508} C_VEL
LIN {X 0,Y 264.276,Z 375.274,A -85,B 0,C 180,E1 -18035.807,E2 -18035.807} C_VEL
LIN {X 0,Y 264.886,Z 378.591,A -85,B 0,C 180,E1 -18039.698,E2 -18039.698} C_VEL
LIN {X 0,Y 265.41,Z 382.112,A -85,B 0,C 180,E1 -18043.509,E2 -18043.509} C_VEL
LIN {X 0,Y 265.697,Z 385.098,A -85,B 0,C 180,E1 -18046.55,E2 -18046.55} C_VEL
LIN {X 0,Y 265.464,Z 387.948,A -85,B 0,C 180,E1 -18049.206,E2 -18049.206} C_VEL
LIN {X 0,Y 266.395,Z 391.062,A -85,B 0,C 180,E1 -18049.494,E2 -18049.494} C_VEL
LIN {X 0,Y 267.497,Z 393.483,A -85,B 0,C 180,E1 -18049.791,E2 -18049.791} C_VEL
LIN {X 0,Y 272.096,Z 405.341,A -85,B 0,C 180,E1 -18051.161,E2 -18051.161} C_VEL
LIN {X 0,Y 276.231,Z 419.009,A -85,B 0,C 180,E1 -18052.754,E2 -18052.754} C_VEL
LIN {X 0,Y 279.088,Z 431.991,A -85,B 0,C 180,E1 -18054.303,E2 -18054.303} C_VEL
LIN {X 0,Y 281.132,Z 446.006,A -85,B 0,C 180,E1 -18056.078,E2 -18056.078} C_VEL
LIN {X 0,Y 282.051,Z 459.304,A -85,B 0,C 180,E1 -18057.907,E2 -18057.907} C_VEL
LIN {X 0,Y 282.03,Z 461.226,A -85,B 0,C 180,E1 -18058.183,E2 -18058.183} C_VEL
LIN {X 0,Y 278.721,Z 474.545,A -85,B 0,C 180,E1 -18059.925,E2 -18059.925} C_VEL
LIN {X 0,Y 275.467,Z 486.418,A -85,B 0,C 180,E1 -18061.837,E2 -18061.837} C_VEL
LIN {X 0,Y 272.368,Z 497.313,A -85,B 0,C 180,E1 -18063.983,E2 -18063.983} C_VEL
LIN {X 0,Y 269.377,Z 507.948,A -85,B 0,C 180,E1 -18066.557,E2 -18066.557} C_VEL
LIN {X 0,Y 266.714,Z 516.793,A -85,B 0,C 180,E1 -18069.163,E2 -18069.163} C_VEL
LIN {X 0,Y 264.978,Z 523.217,A -85,B 0,C 180,E1 -18071.442,E2 -18071.442} C_VEL
LIN {X 0,Y 263.18,Z 530.28,A -85,B 0,C 180,E1 -18074.512,E2 -18074.512} C_VEL
LIN {X 0,Y 261.998,Z 535.847,A -85,B 0,C 180,E1 -18077.609,E2 -18077.609} C_VEL
LIN {X 0,Y 261.347,Z 540.068,A -85,B 0,C 180,E1 -18080.715,E2 -18080.715} C_VEL
LIN {X 0,Y 261.15,Z 543.04,A -85,B 0,C 180,E1 -18083.821,E2 -18083.821} C_VEL
LIN {X 0,Y 261.185,Z 544.817,A -85,B 0,C 180,E1 -18086.916,E2 -18086.916} C_VEL
LIN {X 0,Y 261.248,Z 545.426,A -85,B 0,C 180,E1 -18090.001,E2 -18090.001} C_VEL
LIN {X 0,Y 261.191,Z 544.806,A -85,B 0,C 180,E1 -18093.086,E2 -18093.086} C_VEL
LIN {X 0,Y 261.217,Z 543.017,A -85,B 0,C 180,E1 -18096.179,E2 -18096.179} C_VEL
LIN {X 0,Y 261.348,Z 540.033,A -85,B 0,C 180,E1 -18099.286,E2 -18099.286} C_VEL
LIN {X 0,Y 262,Z 535.804,A -85,B 0,C 180,E1 -18102.392,E2 -18102.392} C_VEL
LIN {X 0,Y 263.188,Z 530.219,A -85,B 0,C 180,E1 -18105.488,E2 -18105.488} C_VEL
LIN {X 0,Y 264.979,Z 523.133,A -85,B 0,C 180,E1 -18108.559,E2 -18108.559} C_VEL
LIN {X 0,Y 267.079,Z 515.568,A -85,B 0,C 180,E1 -18111.213,E2 -18111.213} C_VEL
LIN {X 0,Y 269.774,Z 506.466,A -85,B 0,C 180,E1 -18113.816,E2 -18113.816} C_VEL
LIN {X 0,Y 272.887,Z 495.536,A -85,B 0,C 180,E1 -18116.377,E2 -18116.377} C_VEL
LIN {X 0,Y 276.34,Z 483.266,A -85,B 0,C 180,E1 -18118.688,E2 -18118.688} C_VEL
LIN {X 0,Y 279.735,Z 470.773,A -85,B 0,C 180,E1 -18120.582,E2 -18120.582} C_VEL
LIN {X 0,Y 282.005,Z 461.078,A -85,B 0,C 180,E1 -18121.808,E2 -18121.808} C_VEL
LIN {X 0,Y 281.332,Z 448.576,A -85,B 0,C 180,E1 -18123.552,E2 -18123.552} C_VEL
LIN {X 0,Y 279.868,Z 436.664,A -85,B 0,C 180,E1 -18125.095,E2 -18125.095} C_VEL
LIN {X 0,Y 277.116,Z 422.818,A -85,B 0,C 180,E1 -18126.77,E2 -18126.77} C_VEL
LIN {X 0,Y 273.136,Z 408.513,A -85,B 0,C 180,E1 -18128.425,E2 -18128.425} C_VEL
LIN {X 0,Y 268.42,Z 395.822,A -85,B 0,C 180,E1 -18129.904,E2 -18129.904} C_VEL
LIN {X 0,Y 266.396,Z 391.141,A -85,B 0,C 180,E1 -18130.455,E2 -18130.455} C_VEL
LIN {X 0,Y 265.421,Z 387.861,A -85,B 0,C 180,E1 -18130.765,E2 -18130.765} C_VEL
LIN {X 0,Y 265.731,Z 385.055,A -85,B 0,C 180,E1 -18133.445,E2 -18133.445} C_VEL
LIN {X 0,Y 265.411,Z 382.062,A -85,B 0,C 180,E1 -18136.491,E2 -18136.491} C_VEL
LIN {X 0,Y 264.828,Z 378.386,A -85,B 0,C 180,E1 -18140.438,E2 -18140.438} C_VEL
LIN {X 0,Y 264.278,Z 375.196,A -85,B 0,C 180,E1 -18144.194,E2 -18144.194} C_VEL
LIN {X 0,Y 263.728,Z 371.847,A -85,B 0,C 180,E1 -18148.514,E2 -18148.514} C_VEL
LIN {X 0,Y 263.259,Z 368.721,A -85,B 0,C 180,E1 -18153.01,E2 -18153.01} C_VEL
LIN {X 0,Y 263.229,Z 368.323,A -85,B 0,C 180,E1 -18155.201,E2 -18155.201} C_VEL
LIN {X 0,Y 263.267,Z 368.317,A -85,B 0,C 180,E1 -18159.694,E2 -18159.694} C_VEL
LIN {X 0,Y 263.354,Z 368.309,A -85,B 0,C 180,E1 -18164.522,E2 -18164.522} C_VEL
LIN {X 0,Y 263.378,Z 368.309,A -85,B 0,C 180,E1 -18169.235,E2 -18169.235} C_VEL
LIN {X 0,Y 263.576,Z 368.282,A -85,B 0,C 180,E1 -18172.339,E2 -18172.339} C_VEL
LIN {X 0,Y 263.755,Z 368.256,A -85,B 0,C 180,E1 -18178.473,E2 -18178.473} C_VEL
LIN {X 0,Y 263.756,Z 368.257,A -85,B 0,C 180,E1 -18181.527,E2 -18181.527} C_VEL
LIN {X 0,Y 263.577,Z 368.274,A -85,B 0,C 180,E1 -18187.662,E2 -18187.662} C_VEL
LIN {X 0,Y 263.378,Z 368.288,A -85,B 0,C 180,E1 -18190.766,E2 -18190.766} C_VEL
LIN {X 0,Y 263.354,Z 368.299,A -85,B 0,C 180,E1 -18195.478,E2 -18195.478} C_VEL
LIN {X 0,Y 263.266,Z 368.284,A -85,B 0,C 180,E1 -18200.307,E2 -18200.307} C_VEL
LIN {X 0,Y 263.196,Z 368.316,A -85,B 0,C 180,E1 -18205.293,E2 -18205.293} C_VEL
LIN {X 0,Y 263.169,Z 368.313,A -85,B 0,C 180,E1 -18208.731,E2 -18208.731} C_VEL
LIN {X 0,Y 263.136,Z 368.318,A -85,B 0,C 180,E1 -18212.288,E2 -18212.288} C_VEL
LIN {X 0,Y 263.191,Z 368.327,A -85,B 0,C 180,E1 -18215.978,E2 -18215.978} C_VEL
LIN {X 0,Y 263.118,Z 368.335,A -85,B 0,C 180,E1 -18219.87,E2 -18219.87} C_VEL
LIN {X 0,Y 263.1,Z 368.343,A -85,B 0,C 180,E1 -18223.989,E2 -18223.989} C_VEL
LIN {X 0,Y 263.064,Z 368.348,A -85,B 0,C 180,E1 -18226.165,E2 -18226.165} C_VEL
LIN {X 0,Y 263.115,Z 369.472,A -85,B 0,C 180,E1 -18228.896,E2 -18228.896} C_VEL
LIN {X 0,Y 264.183,Z 372.296,A -85,B 0,C 180,E1 -18229.217,E2 -18229.217} C_VEL
LIN {X 0,Y 265.813,Z 374.87,A -85,B 0,C 180,E1 -18229.631,E2 -18229.631} C_VEL
LIN {X 0,Y 271.925,Z 386.647,A -85,B 0,C 180,E1 -18231.354,E2 -18231.354} C_VEL
LIN {X 0,Y 276.961,Z 398.236,A -85,B 0,C 180,E1 -18233.015,E2 -18233.015} C_VEL
LIN {X 0,Y 281.043,Z 410.21,A -85,B 0,C 180,E1 -18234.727,E2 -18234.727} C_VEL
LIN {X 0,Y 284.33,Z 423.013,A -85,B 0,C 180,E1 -18236.6,E2 -18236.6} C_VEL
LIN {X 0,Y 285.543,Z 429.943,A -85,B 0,C 180,E1 -18237.639,E2 -18237.639} C_VEL
LIN {X 0,Y 282.718,Z 442.92,A -85,B 0,C 180,E1 -18239.155,E2 -18239.155} C_VEL
LIN {X 0,Y 279.759,Z 454.902,A -85,B 0,C 180,E1 -18240.873,E2 -18240.873} C_VEL
LIN {X 0,Y 276.745,Z 465.963,A -85,B 0,C 180,E1 -18242.798,E2 -18242.798} C_VEL
LIN {X 0,Y 273.862,Z 476.101,A -85,B 0,C 180,E1 -18244.948,E2 -18244.948} C_VEL
LIN {X 0,Y 270.851,Z 486.014,A -85,B 0,C 180,E1 -18247.496,E2 -18247.496} C_VEL
LIN {X 0,Y 268.264,Z 494.228,A -85,B 0,C 180,E1 -18250.087,E2 -18250.087} C_VEL
LIN {X 0,Y 266.459,Z 500.147,A -85,B 0,C 180,E1 -18252.342,E2 -18252.342} C_VEL
LIN {X 0,Y 264.474,Z 506.654,A -85,B 0,C 180,E1 -18255.377,E2 -18255.377} C_VEL
LIN {X 0,Y 263.13,Z 511.727,A -85,B 0,C 180,E1 -18258.444,E2 -18258.444} C_VEL
LIN {X 0,Y 262.32,Z 514.65,A -85,B 0,C 180,E1 -18260.749,E2 -18260.749} C_VEL
LIN {X 0,Y 261.729,Z 517.502,A -85,B 0,C 180,E1 -18263.833,E2 -18263.833} C_VEL
LIN {X 0,Y 261.418,Z 519.215,A -85,B 0,C 180,E1 -18266.917,E2 -18266.917} C_VEL
LIN {X 0,Y 261.292,Z 519.813,A -85,B 0,C 180,E1 -18269.999,E2 -18269.999} C_VEL
LIN {X 0,Y 261.417,Z 519.253,A -85,B 0,C 180,E1 -18273.082,E2 -18273.082} C_VEL
LIN {X 0,Y 261.728,Z 517.592,A -85,B 0,C 180,E1 -18276.165,E2 -18276.165} C_VEL
LIN {X 0,Y 262.311,Z 514.788,A -85,B 0,C 180,E1 -18279.25,E2 -18279.25} C_VEL
LIN {X 0,Y 263.374,Z 510.764,A -85,B 0,C 180,E1 -18282.325,E2 -18282.325} C_VEL
LIN {X 0,Y 264.883,Z 505.422,A -85,B 0,C 180,E1 -18285.386,E2 -18285.386} C_VEL
LIN {X 0,Y 266.41,Z 500.427,A -85,B 0,C 180,E1 -18287.66,E2 -18287.66} C_VEL
LIN {X 0,Y 268.508,Z 493.472,A -85,B 0,C 180,E1 -18290.292,E2 -18290.292} C_VEL
LIN {X 0,Y 271.203,Z 485.085,A -85,B 0,C 180,E1 -18292.874,E2 -18292.874} C_VEL
LIN {X 0,Y 274.218,Z 474.982,A -85,B 0,C 180,E1 -18295.422,E2 -18295.422} C_VEL
LIN {X 0,Y 277.408,Z 463.768,A -85,B 0,C 180,E1 -18297.722,E2 -18297.722} C_VEL
LIN {X 0,Y 280.541,Z 452.201,A -85,B 0,C 180,E1 -18299.654,E2 -18299.654} C_VEL
LIN {X 0,Y 283.5,Z 439.708,A -85,B 0,C 180,E1 -18301.371,E2 -18301.371} C_VEL
LIN {X 0,Y 285.526,Z 430.375,A -85,B 0,C 180,E1 -18302.431,E2 -18302.431} C_VEL
LIN {X 0,Y 285.032,Z 426.253,A -85,B 0,C 180,E1 -18303.035,E2 -18303.035} C_VEL
LIN {X 0,Y 281.935,Z 413.123,A -85,B 0,C 180,E1 -18304.983,E2 -18304.983} C_VEL
LIN {X 0,Y 277.727,Z 400.311,A -85,B 0,C 180,E1 -18306.823,E2 -18306.823} C_VEL
LIN {X 0,Y 272.821,Z 388.496,A -85,B 0,C 180,E1 -18308.505,E2 -18308.505} C_VEL
LIN {X 0,Y 267.148,Z 377.277,A -85,B 0,C 180,E1 -18310.158,E2 -18310.158} C_VEL
LIN {X 0,Y 264.974,Z 373.405,A -85,B 0,C 180,E1 -18310.726,E2 -18310.726} C_VEL
LIN {X 0,Y 263.445,Z 370.673,A -85,B 0,C 180,E1 -18311.133,E2 -18311.133} C_VEL
LIN {X 0,Y 263.125,Z 369.395,A -85,B 0,C 180,E1 -18311.262,E2 -18311.262} C_VEL
LIN {X 0,Y 263.062,Z 368.339,A -85,B 0,C 180,E1 -18313.996,E2 -18313.996} C_VEL
LIN {X 0,Y 263.122,Z 368.335,A -85,B 0,C 180,E1 -18318.106,E2 -18318.106} C_VEL
LIN {X 0,Y 263.164,Z 368.331,A -85,B 0,C 180,E1 -18322.104,E2 -18322.104} C_VEL
LIN {X 0,Y 263.182,Z 368.313,A -85,B 0,C 180,E1 -18325.89,E2 -18325.89} C_VEL
LIN {X 0,Y 263.149,Z 368.331,A -85,B 0,C 180,E1 -18329.506,E2 -18329.506} C_VEL
LIN {X 0,Y 263.191,Z 368.302,A -85,B 0,C 180,E1 -18333.002,E2 -18333.002} C_VEL
LIN {X 0,Y 263.183,Z 368.326,A -85,B 0,C 180,E1 -18336.387,E2 -18336.387} C_VEL
LIN {X 0,Y 263.262,Z 368.288,A -85,B 0,C 180,E1 -18339.693,E2 -18339.693} C_VEL
LIN {X 0,Y 263.349,Z 368.298,A -85,B 0,C 180,E1 -18344.522,E2 -18344.522} C_VEL
LIN {X 0,Y 263.373,Z 368.296,A -85,B 0,C 180,E1 -18349.234,E2 -18349.234} C_VEL
LIN {X 0,Y 263.571,Z 368.278,A -85,B 0,C 180,E1 -18352.338,E2 -18352.338} C_VEL
LIN {X 0,Y 263.75,Z 368.257,A -85,B 0,C 180,E1 -18358.473,E2 -18358.473} C_VEL
LIN {X 0,Y 263.75,Z 368.259,A -85,B 0,C 180,E1 -18361.527,E2 -18361.527} C_VEL
LIN {X 0,Y 263.571,Z 368.28,A -85,B 0,C 180,E1 -18367.661,E2 -18367.661} C_VEL
LIN {X 0,Y 263.372,Z 368.305,A -85,B 0,C 180,E1 -18370.766,E2 -18370.766} C_VEL
LIN {X 0,Y 263.348,Z 368.3,A -85,B 0,C 180,E1 -18375.478,E2 -18375.478} C_VEL
LIN {X 0,Y 263.232,Z 368.316,A -85,B 0,C 180,E1 -18377.85,E2 -18377.85} C_VEL
LIN {X 0,Y 262.552,Z 368.405,A -85,B 0,C 180,E1 -18379.126,E2 -18379.126} C_VEL
LIN {X 0,Y 259.68,Z 368.762,A -85,B 0,C 180,E1 -18381.206,E2 -18381.206} C_VEL
LIN {X 0,Y 257.26,Z 369.068,A -85,B 0,C 180,E1 -18382.897,E2 -18382.897} C_VEL
LIN {X 0,Y 256.24,Z 369.195,A -85,B 0,C 180,E1 -18384.209,E2 -18384.209} C_VEL
LIN {X 0,Y 256.167,Z 369.203,A -85,B 0,C 180,E1 -18384.653,E2 -18384.653} C_VEL
LIN {X 0,Y 256.222,Z 369.636,A -85,B 0,C 180,E1 -18386.032,E2 -18386.032} C_VEL
LIN {X 0,Y 256.563,Z 371.925,A -85,B 0,C 180,E1 -18389.542,E2 -18389.542} C_VEL
LIN {X 0,Y 256.964,Z 374.537,A -85,B 0,C 180,E1 -18393.161,E2 -18393.161} C_VEL
LIN {X 0,Y 257.561,Z 378.12,A -85,B 0,C 180,E1 -18397.693,E2 -18397.693} C_VEL
LIN {X 0,Y 258.022,Z 380.803,A -85,B 0,C 180,E1 -18400.822,E2 -18400.822} C_VEL
LIN {X 0,Y 258.561,Z 384.642,A -85,B 0,C 180,E1 -18405.033,E2 -18405.033} C_VEL
LIN {X 0,Y 258.623,Z 387.467,A -85,B 0,C 180,E1 -18407.882,E2 -18407.882} C_VEL
LIN {X 0,Y 259.599,Z 390.707,A -85,B 0,C 180,E1 -18408.203,E2 -18408.203} C_VEL
LIN {X 0,Y 260.783,Z 392.995,A -85,B 0,C 180,E1 -18408.529,E2 -18408.529} C_VEL
LIN {X 0,Y 265.817,Z 406.069,A -85,B 0,C 180,E1 -18410.135,E2 -18410.135} C_VEL
LIN {X 0,Y 269.615,Z 418.196,A -85,B 0,C 180,E1 -18411.645,E2 -18411.645} C_VEL
LIN {X 0,Y 272.669,Z 431.77,A -85,B 0,C 180,E1 -18413.344,E2 -18413.344} C_VEL
LIN {X 0,Y 274.67,Z 445.34,A -85,B 0,C 180,E1 -18415.131,E2 -18415.131} C_VEL
LIN {X 0,Y 275.566,Z 458.653,A -85,B 0,C 180,E1 -18417.016,E2 -18417.016} C_VEL
LIN {X 0,Y 275.409,Z 463.58,A -85,B 0,C 180,E1 -18417.733,E2 -18417.733} C_VEL
LIN {X 0,Y 271.897,Z 476.558,A -85,B 0,C 180,E1 -18419.519,E2 -18419.519} C_VEL
LIN {X 0,Y 268.593,Z 488.036,A -85,B 0,C 180,E1 -18421.477,E2 -18421.477} C_VEL
LIN {X 0,Y 265.457,Z 498.607,A -85,B 0,C 180,E1 -18423.676,E2 -18423.676} C_VEL
LIN {X 0,Y 262.713,Z 507.763,A -85,B 0,C 180,E1 -18425.977,E2 -18425.977} C_VEL
LIN {X 0,Y 260.036,Z 516.443,A -85,B 0,C 180,E1 -18428.601,E2 -18428.601} C_VEL
LIN {X 0,Y 258.156,Z 522.866,A -85,B 0,C 180,E1 -18430.933,E2 -18430.933} C_VEL
LIN {X 0,Y 256.257,Z 529.928,A -85,B 0,C 180,E1 -18434.083,E2 -18434.083} C_VEL
LIN {X 0,Y 255.013,Z 535.497,A -85,B 0,C 180,E1 -18437.264,E2 -18437.264} C_VEL
LIN {X 0,Y 254.283,Z 539.718,A -85,B 0,C 180,E1 -18440.455,E2 -18440.455} C_VEL
LIN {X 0,Y 254.05,Z 542.69,A -85,B 0,C 180,E1 -18443.648,E2 -18443.648} C_VEL
LIN {X 0,Y 254.096,Z 544.469,A -85,B 0,C 180,E1 -18446.83,E2 -18446.83} C_VEL
LIN {X 0,Y 254.17,Z 545.079,A -85,B 0,C 180,E1 -18450.001,E2 -18450.001} C_VEL
LIN {X 0,Y 254.103,Z 544.458,A -85,B 0,C 180,E1 -18453.172,E2 -18453.172} C_VEL
LIN {X 0,Y 254.14,Z 542.668,A -85,B 0,C 180,E1 -18456.352,E2 -18456.352} C_VEL
LIN {X 0,Y 254.285,Z 539.681,A -85,B 0,C 180,E1 -18459.546,E2 -18459.546} C_VEL
LIN {X 0,Y 255.015,Z 535.452,A -85,B 0,C 180,E1 -18462.737,E2 -18462.737} C_VEL
LIN {X 0,Y 256.265,Z 529.866,A -85,B 0,C 180,E1 -18465.918,E2 -18465.918} C_VEL
LIN {X 0,Y 258.156,Z 522.778,A -85,B 0,C 180,E1 -18469.068,E2 -18469.068} C_VEL
LIN {X 0,Y 260.399,Z 515.214,A -85,B 0,C 180,E1 -18471.784,E2 -18471.784} C_VEL
LIN {X 0,Y 263.169,Z 506.316,A -85,B 0,C 180,E1 -18474.39,E2 -18474.39} C_VEL
LIN {X 0,Y 265.96,Z 496.829,A -85,B 0,C 180,E1 -18476.695,E2 -18476.695} C_VEL
LIN {X 0,Y 269.202,Z 485.911,A -85,B 0,C 180,E1 -18478.881,E2 -18478.881} C_VEL
LIN {X 0,Y 272.577,Z 474.009,A -85,B 0,C 180,E1 -18480.828,E2 -18480.828} C_VEL
LIN {X 0,Y 275.579,Z 462.436,A -85,B 0,C 180,E1 -18482.382,E2 -18482.382} C_VEL
LIN {X 0,Y 275.064,Z 449.982,A -85,B 0,C 180,E1 -18484.202,E2 -18484.202} C_VEL
LIN {X 0,Y 273.341,Z 436.042,A -85,B 0,C 180,E1 -18486.086,E2 -18486.086} C_VEL
LIN {X 0,Y 270.845,Z 423.434,A -85,B 0,C 180,E1 -18487.678,E2 -18487.678} C_VEL
LIN {X 0,Y 267.25,Z 410.412,A -85,B 0,C 180,E1 -18489.284,E2 -18489.284} C_VEL
LIN {X 0,Y 263.18,Z 399.094,A -85,B 0,C 180,E1 -18490.686,E2 -18490.686} C_VEL
LIN {X 0,Y 260.164,Z 391.735,A -85,B 0,C 180,E1 -18491.593,E2 -18491.593} C_VEL
LIN {X 0,Y 258.824,Z 388.563,A -85,B 0,C 180,E1 -18491.986,E2 -18491.986} C_VEL
LIN {X 0,Y 258.62,Z 387.464,A -85,B 0,C 180,E1 -18492.081,E2 -18492.081} C_VEL
LIN {X 0,Y 258.599,Z 384.546,A -85,B 0,C 180,E1 -18495.041,E2 -18495.041} C_VEL
LIN {X 0,Y 258.018,Z 380.732,A -85,B 0,C 180,E1 -18499.177,E2 -18499.177} C_VEL
LIN {X 0,Y 257.462,Z 377.377,A -85,B 0,C 180,E1 -18503.092,E2 -18503.092} C_VEL
LIN {X 0,Y 256.948,Z 374.422,A -85,B 0,C 180,E1 -18506.836,E2 -18506.836} C_VEL
LIN {X 0,Y 256.491,Z 371.318,A -85,B 0,C 180,E1 -18511.262,E2 -18511.262} C_VEL
LIN {X 0,Y 256.191,Z 369.199,A -85,B 0,C 180,E1 -18514.862,E2 -18514.862} C_VEL
LIN {X 0,Y 256.17,Z 369.202,A -85,B 0,C 180,E1 -18519.105,E2 -18519.105} C_VEL
LIN {X 0,Y 256.303,Z 369.188,A -85,B 0,C 180,E1 -18524.085,E2 -18524.085} C_VEL
LIN {X 0,Y 256.313,Z 369.188,A -85,B 0,C 180,E1 -18528.934,E2 -18528.934} C_VEL
LIN {X 0,Y 256.544,Z 369.159,A -85,B 0,C 180,E1 -18532.127,E2 -18532.127} C_VEL
LIN {X 0,Y 256.718,Z 369.133,A -85,B 0,C 180,E1 -18538.431,E2 -18538.431} C_VEL
LIN {X 0,Y 256.718,Z 369.133,A -85,B 0,C 180,E1 -18541.569,E2 -18541.569} C_VEL
LIN {X 0,Y 256.544,Z 369.152,A -85,B 0,C 180,E1 -18547.873,E2 -18547.873} C_VEL
LIN {X 0,Y 256.313,Z 369.161,A -85,B 0,C 180,E1 -18551.066,E2 -18551.066} C_VEL
LIN {X 0,Y 256.304,Z 369.181,A -85,B 0,C 180,E1 -18555.915,E2 -18555.915} C_VEL
LIN {X 0,Y 256.166,Z 369.169,A -85,B 0,C 180,E1 -18560.895,E2 -18560.895} C_VEL
LIN {X 0,Y 256.174,Z 369.193,A -85,B 0,C 180,E1 -18565.13,E2 -18565.13} C_VEL
LIN {X 0,Y 256.107,Z 369.204,A -85,B 0,C 180,E1 -18569.601,E2 -18569.601} C_VEL
LIN {X 0,Y 256.088,Z 369.189,A -85,B 0,C 180,E1 -18573.29,E2 -18573.29} C_VEL
LIN {X 0,Y 256.132,Z 369.206,A -85,B 0,C 180,E1 -18577.275,E2 -18577.275} C_VEL
LIN {X 0,Y 256.06,Z 369.215,A -85,B 0,C 180,E1 -18581.203,E2 -18581.203} C_VEL
LIN {X 0,Y 256.015,Z 369.226,A -85,B 0,C 180,E1 -18585.54,E2 -18585.54} C_VEL
LIN {X 0,Y 256.043,Z 369.873,A -85,B 0,C 180,E1 -18587.497,E2 -18587.497} C_VEL
LIN {X 0,Y 256.978,Z 372.561,A -85,B 0,C 180,E1 -18587.806,E2 -18587.806} C_VEL
LIN {X 0,Y 258.937,Z 375.339,A -85,B 0,C 180,E1 -18588.325,E2 -18588.325} C_VEL
LIN {X 0,Y 265.261,Z 387.258,A -85,B 0,C 180,E1 -18590.206,E2 -18590.206} C_VEL
LIN {X 0,Y 270.333,Z 398.823,A -85,B 0,C 180,E1 -18591.963,E2 -18591.963} C_VEL
LIN {X 0,Y 274.482,Z 410.708,A -85,B 0,C 180,E1 -18593.761,E2 -18593.761} C_VEL
LIN {X 0,Y 277.597,Z 422.27,A -85,B 0,C 180,E1 -18595.533,E2 -18595.533} C_VEL
LIN {X 0,Y 279.336,Z 431.405,A -85,B 0,C 180,E1 -18596.98,E2 -18596.98} C_VEL
LIN {X 0,Y 276.37,Z 444.553,A -85,B 0,C 180,E1 -18598.579,E2 -18598.579} C_VEL
LIN {X 0,Y 272.981,Z 457.374,A -85,B 0,C 180,E1 -18600.502,E2 -18600.502} C_VEL
LIN {X 0,Y 270.051,Z 467.745,A -85,B 0,C 180,E1 -18602.407,E2 -18602.407} C_VEL
LIN {X 0,Y 266.979,Z 477.97,A -85,B 0,C 180,E1 -18604.673,E2 -18604.673} C_VEL
LIN {X 0,Y 263.886,Z 487.622,A -85,B 0,C 180,E1 -18607.283,E2 -18607.283} C_VEL
LIN {X 0,Y 261.242,Z 495.66,A -85,B 0,C 180,E1 -18609.94,E2 -18609.94} C_VEL
LIN {X 0,Y 259.15,Z 502.279,A -85,B 0,C 180,E1 -18612.643,E2 -18612.643} C_VEL
LIN {X 0,Y 257.152,Z 508.405,A -85,B 0,C 180,E1 -18615.76,E2 -18615.76} C_VEL
LIN {X 0,Y 255.865,Z 513.12,A -85,B 0,C 180,E1 -18618.914,E2 -18618.914} C_VEL
LIN {X 0,Y 254.949,Z 516.571,A -85,B 0,C 180,E1 -18622.077,E2 -18622.077} C_VEL
LIN {X 0,Y 254.501,Z 518.844,A -85,B 0,C 180,E1 -18625.247,E2 -18625.247} C_VEL
LIN {X 0,Y 254.24,Z 520.005,A -85,B 0,C 180,E1 -18628.415,E2 -18628.415} C_VEL
LIN {X 0,Y 254.239,Z 520.018,A -85,B 0,C 180,E1 -18631.583,E2 -18631.583} C_VEL
LIN {X 0,Y 254.5,Z 518.908,A -85,B 0,C 180,E1 -18634.751,E2 -18634.751} C_VEL
LIN {X 0,Y 254.947,Z 516.685,A -85,B 0,C 180,E1 -18637.922,E2 -18637.922} C_VEL
LIN {X 0,Y 255.833,Z 513.28,A -85,B 0,C 180,E1 -18641.086,E2 -18641.086} C_VEL
LIN {X 0,Y 257.102,Z 508.617,A -85,B 0,C 180,E1 -18644.241,E2 -18644.241} C_VEL
LIN {X 0,Y 259.105,Z 502.554,A -85,B 0,C 180,E1 -18647.359,E2 -18647.359} C_VEL
LIN {X 0,Y 261.151,Z 495.972,A -85,B 0,C 180,E1 -18650.066,E2 -18650.066} C_VEL
LIN {X 0,Y 263.823,Z 487.992,A -85,B 0,C 180,E1 -18652.722,E2 -18652.722} C_VEL
LIN {X 0,Y 266.857,Z 478.416,A -85,B 0,C 180,E1 -18655.338,E2 -18655.338} C_VEL
LIN {X 0,Y 269.763,Z 468.854,A -85,B 0,C 180,E1 -18657.486,E2 -18657.486} C_VEL
LIN {X 0,Y 273.145,Z 456.944,A -85,B 0,C 180,E1 -18659.689,E2 -18659.689} C_VEL
LIN {X 0,Y 276.231,Z 445.313,A -85,B 0,C 180,E1 -18661.437,E2 -18661.437} C_VEL
LIN {X 0,Y 279.093,Z 433.071,A -85,B 0,C 180,E1 -18662.951,E2 -18662.951} C_VEL
LIN {X 0,Y 279.337,Z 431.85,A -85,B 0,C 180,E1 -18663.086,E2 -18663.086} C_VEL
LIN {X 0,Y 277.505,Z 421.881,A -85,B 0,C 180,E1 -18664.66,E2 -18664.66} C_VEL
LIN {X 0,Y 274.666,Z 411.191,A -85,B 0,C 180,E1 -18666.291,E2 -18666.291} C_VEL
LIN {X 0,Y 270.315,Z 398.676,A -85,B 0,C 180,E1 -18668.185,E2 -18668.185} C_VEL
LIN {X 0,Y 265.013,Z 386.55,A -85,B 0,C 180,E1 -18670.026,E2 -18670.026} C_VEL
LIN {X 0,Y 260.133,Z 377.519,A -85,B 0,C 180,E1 -18671.485,E2 -18671.485} C_VEL
LIN {X 0,Y 258.207,Z 374.166,A -85,B 0,C 180,E1 -18672.017,E2 -18672.017} C_VEL
LIN {X 0,Y 256.485,Z 371.511,A -85,B 0,C 180,E1 -18672.487,E2 -18672.487} C_VEL
LIN {X 0,Y 256.041,Z 369.836,A -85,B 0,C 180,E1 -18672.665,E2 -18672.665} C_VEL
LIN {X 0,Y 256.011,Z 369.218,A -85,B 0,C 180,E1 -18674.459,E2 -18674.459} C_VEL
LIN {X 0,Y 256.055,Z 369.217,A -85,B 0,C 180,E1 -18678.796,E2 -18678.796} C_VEL
LIN {X 0,Y 256.143,Z 369.203,A -85,B 0,C 180,E1 -18682.869,E2 -18682.869} C_VEL
LIN {X 0,Y 256.084,Z 369.191,A -85,B 0,C 180,E1 -18686.709,E2 -18686.709} C_VEL
LIN {X 0,Y 256.136,Z 369.191,A -85,B 0,C 180,E1 -18691.404,E2 -18691.404} C_VEL
LIN {X 0,Y 256.166,Z 369.2,A -85,B 0,C 180,E1 -18695.699,E2 -18695.699} C_VEL
LIN {X 0,Y 256.164,Z 369.172,A -85,B 0,C 180,E1 -18699.105,E2 -18699.105} C_VEL
LIN {X 0,Y 256.298,Z 369.181,A -85,B 0,C 180,E1 -18704.085,E2 -18704.085} C_VEL
LIN {X 0,Y 256.308,Z 369.169,A -85,B 0,C 180,E1 -18708.934,E2 -18708.934} C_VEL
LIN {X 0,Y 256.538,Z 369.153,A -85,B 0,C 180,E1 -18712.127,E2 -18712.127} C_VEL
LIN {X 0,Y 256.713,Z 369.133,A -85,B 0,C 180,E1 -18718.431,E2 -18718.431} C_VEL
LIN {X 0,Y 256.713,Z 369.136,A -85,B 0,C 180,E1 -18721.569,E2 -18721.569} C_VEL
LIN {X 0,Y 256.538,Z 369.155,A -85,B 0,C 180,E1 -18727.873,E2 -18727.873} C_VEL
LIN {X 0,Y 256.308,Z 369.184,A -85,B 0,C 180,E1 -18731.066,E2 -18731.066} C_VEL
LIN {X 0,Y 256.298,Z 369.179,A -85,B 0,C 180,E1 -18735.915,E2 -18735.915} C_VEL
LIN {X 0,Y 256.164,Z 369.199,A -85,B 0,C 180,E1 -18740.895,E2 -18740.895} C_VEL
LIN {X 0,Y 256.167,Z 369.203,A -85,B 0,C 180,E1 -18744.653,E2 -18744.653} C_VEL
LIN {X 0,Y 255.886,Z 369.474,A -85,B 0,C 180,E1 -18745.531,E2 -18745.531} C_VEL
LIN {X 0,Y 254.087,Z 370.865,A -85,B 0,C 180,E1 -18747.24,E2 -18747.24} C_VEL
LIN {X 0,Y 250.681,Z 373.317,A -85,B 0,C 180,E1 -18749.793,E2 -18749.793} C_VEL
LIN {X 0,Y 249.812,Z 374.409,A -85,B 0,C 180,E1 -18751.124,E2 -18751.124} C_VEL
LIN {X 0,Y 249.787,Z 374.737,A -85,B 0,C 180,E1 -18751.574,E2 -18751.574} C_VEL
LIN {X 0,Y 250.359,Z 378.107,A -85,B 0,C 180,E1 -18756.122,E2 -18756.122} C_VEL
LIN {X 0,Y 251.036,Z 382.026,A -85,B 0,C 180,E1 -18760.898,E2 -18760.898} C_VEL
LIN {X 0,Y 251.444,Z 385.049,A -85,B 0,C 180,E1 -18764.328,E2 -18764.328} C_VEL
LIN {X 0,Y 251.647,Z 387.155,A -85,B 0,C 180,E1 -18766.434,E2 -18766.434} C_VEL
LIN {X 0,Y 252.629,Z 390.151,A -85,B 0,C 180,E1 -18766.768,E2 -18766.768} C_VEL
LIN {X 0,Y 254.03,Z 392.503,A -85,B 0,C 180,E1 -18767.166,E2 -18767.166} C_VEL
LIN {X 0,Y 258.069,Z 402.55,A -85,B 0,C 180,E1 -18768.496,E2 -18768.496} C_VEL
LIN {X 0,Y 262.236,Z 414.773,A -85,B 0,C 180,E1 -18770.117,E2 -18770.117} C_VEL
LIN {X 0,Y 265.45,Z 427.529,A -85,B 0,C 180,E1 -18771.782,E2 -18771.782} C_VEL
LIN {X 0,Y 267.423,Z 438.559,A -85,B 0,C 180,E1 -18773.277,E2 -18773.277} C_VEL
LIN {X 0,Y 268.817,Z 451.121,A -85,B 0,C 180,E1 -18775.054,E2 -18775.054} C_VEL
LIN {X 0,Y 269.259,Z 463.226,A -85,B 0,C 180,E1 -18776.903,E2 -18776.903} C_VEL
LIN {X 0,Y 266.131,Z 475.033,A -85,B 0,C 180,E1 -18778.564,E2 -18778.564} C_VEL
LIN {X 0,Y 262.965,Z 485.724,A -85,B 0,C 180,E1 -18780.369,E2 -18780.369} C_VEL
LIN {X 0,Y 259.553,Z 496.615,A -85,B 0,C 180,E1 -18782.593,E2 -18782.593} C_VEL
LIN {X 0,Y 256.326,Z 506.861,A -85,B 0,C 180,E1 -18785.165,E2 -18785.165} C_VEL
LIN {X 0,Y 253.782,Z 514.963,A -85,B 0,C 180,E1 -18787.619,E2 -18787.619} C_VEL
LIN {X 0,Y 251.368,Z 522.515,A -85,B 0,C 180,E1 -18790.397,E2 -18790.397} C_VEL
LIN {X 0,Y 249.355,Z 529.577,A -85,B 0,C 180,E1 -18793.63,E2 -18793.63} C_VEL
LIN {X 0,Y 248.009,Z 535.146,A -85,B 0,C 180,E1 -18796.898,E2 -18796.898} C_VEL
LIN {X 0,Y 247.236,Z 539.368,A -85,B 0,C 180,E1 -18800.18,E2 -18800.18} C_VEL
LIN {X 0,Y 246.961,Z 542.341,A -85,B 0,C 180,E1 -18803.464,E2 -18803.464} C_VEL
LIN {X 0,Y 247.009,Z 544.121,A -85,B 0,C 180,E1 -18806.739,E2 -18806.739} C_VEL
LIN {X 0,Y 247.095,Z 544.732,A -85,B 0,C 180,E1 -18810.001,E2 -18810.001} C_VEL
LIN {X 0,Y 247.017,Z 544.11,A -85,B 0,C 180,E1 -18813.263,E2 -18813.263} C_VEL
LIN {X 0,Y 247.043,Z 542.317,A -85,B 0,C 180,E1 -18816.535,E2 -18816.535} C_VEL
LIN {X 0,Y 247.237,Z 539.33,A -85,B 0,C 180,E1 -18819.821,E2 -18819.821} C_VEL
LIN {X 0,Y 248.011,Z 535.099,A -85,B 0,C 180,E1 -18823.103,E2 -18823.103} C_VEL
LIN {X 0,Y 249.362,Z 529.512,A -85,B 0,C 180,E1 -18826.371,E2 -18826.371} C_VEL
LIN {X 0,Y 251.367,Z 522.424,A -85,B 0,C 180,E1 -18829.604,E2 -18829.604} C_VEL
LIN {X 0,Y 253.769,Z 514.862,A -85,B 0,C 180,E1 -18832.384,E2 -18832.384} C_VEL
LIN {X 0,Y 256.539,Z 506.292,A -85,B 0,C 180,E1 -18834.959,E2 -18834.959} C_VEL
LIN {X 0,Y 259.574,Z 496.475,A -85,B 0,C 180,E1 -18837.406,E2 -18837.406} C_VEL
LIN {X 0,Y 262.95,Z 485.557,A -85,B 0,C 180,E1 -18839.635,E2 -18839.635} C_VEL
LIN {X 0,Y 266.476,Z 473.656,A -85,B 0,C 180,E1 -18841.614,E2 -18841.614} C_VEL
LIN {X 0,Y 269.037,Z 464.486,A -85,B 0,C 180,E1 -18842.89,E2 -18842.89} C_VEL
LIN {X 0,Y 269.098,Z 457.693,A -85,B 0,C 180,E1 -18843.935,E2 -18843.935} C_VEL
LIN {X 0,Y 268.28,Z 445.619,A -85,B 0,C 180,E1 -18845.7,E2 -18845.7} C_VEL
LIN {X 0,Y 266.219,Z 431.607,A -85,B 0,C 180,E1 -18847.629,E2 -18847.629} C_VEL
LIN {X 0,Y 262.911,Z 417.193,A -85,B 0,C 180,E1 -18849.523,E2 -18849.523} C_VEL
LIN {X 0,Y 258.742,Z 404.194,A -85,B 0,C 180,E1 -18851.232,E2 -18851.232} C_VEL
LIN {X 0,Y 255.085,Z 395.221,A -85,B 0,C 180,E1 -18852.444,E2 -18852.444} C_VEL
LIN {X 0,Y 253.361,Z 391.399,A -85,B 0,C 180,E1 -18852.967,E2 -18852.967} C_VEL
LIN {X 0,Y 251.877,Z 388.204,A -85,B 0,C 180,E1 -18853.419,E2 -18853.419} C_VEL
LIN {X 0,Y 251.669,Z 386.979,A -85,B 0,C 180,E1 -18853.568,E2 -18853.568} C_VEL
LIN {X 0,Y 251.317,Z 384.116,A -85,B 0,C 180,E1 -18856.643,E2 -18856.643} C_VEL
LIN {X 0,Y 250.911,Z 381.307,A -85,B 0,C 180,E1 -18859.892,E2 -18859.892} C_VEL
LIN {X 0,Y 250.281,Z 377.529,A -85,B 0,C 180,E1 -18864.522,E2 -18864.522} C_VEL
LIN {X 0,Y 249.862,Z 375.15,A -85,B 0,C 180,E1 -18867.695,E2 -18867.695} C_VEL
LIN {X 0,Y 249.517,Z 372.649,A -85,B 0,C 180,E1 -18871.391,E2 -18871.391} C_VEL
LIN {X 0,Y 249.194,Z 370.432,A -85,B 0,C 180,E1 -18874.973,E2 -18874.973} C_VEL
LIN {X 0,Y 249.098,Z 370.082,A -85,B 0,C 180,E1 -18878.601,E2 -18878.601} C_VEL
LIN {X 0,Y 249.245,Z 370.067,A -85,B 0,C 180,E1 -18883.622,E2 -18883.622} C_VEL
LIN {X 0,Y 249.257,Z 370.067,A -85,B 0,C 180,E1 -18888.617,E2 -18888.617} C_VEL
LIN {X 0,Y 249.488,Z 370.037,A -85,B 0,C 180,E1 -18891.903,E2 -18891.903} C_VEL
LIN {X 0,Y 249.44,Z 370.035,A -85,B 0,C 180,E1 -18896.77,E2 -18896.77} C_VEL
LIN {X 0,Y 249.732,Z 369.998,A -85,B 0,C 180,E1 -18900,E2 -18900} C_VEL
LIN {X 0,Y 249.44,Z 370.033,A -85,B 0,C 180,E1 -18903.231,E2 -18903.231} C_VEL
LIN {X 0,Y 249.488,Z 370.033,A -85,B 0,C 180,E1 -18908.097,E2 -18908.097} C_VEL
LIN {X 0,Y 249.257,Z 370.034,A -85,B 0,C 180,E1 -18911.383,E2 -18911.383} C_VEL
LIN {X 0,Y 249.246,Z 370.062,A -85,B 0,C 180,E1 -18916.378,E2 -18916.378} C_VEL
LIN {X 0,Y 249.088,Z 370.055,A -85,B 0,C 180,E1 -18921.518,E2 -18921.518} C_VEL
LIN {X 0,Y 249.12,Z 370.067,A -85,B 0,C 180,E1 -18925.475,E2 -18925.475} C_VEL
LIN {X 0,Y 249.076,Z 370.071,A -85,B 0,C 180,E1 -18928.989,E2 -18928.989} C_VEL
LIN {X 0,Y 249.039,Z 370.071,A -85,B 0,C 180,E1 -18932.425,E2 -18932.425} C_VEL
LIN {X 0,Y 249.072,Z 370.086,A -85,B 0,C 180,E1 -18936.338,E2 -18936.338} C_VEL
LIN {X 0,Y 249.029,Z 370.092,A -85,B 0,C 180,E1 -18940.474,E2 -18940.474} C_VEL
LIN {X 0,Y 248.97,Z 370.102,A -85,B 0,C 180,E1 -18944.887,E2 -18944.887} C_VEL
LIN {X 0,Y 248.973,Z 370.297,A -85,B 0,C 180,E1 -18945.982,E2 -18945.982} C_VEL
LIN {X 0,Y 249.977,Z 373.094,A -85,B 0,C 180,E1 -18946.336,E2 -18946.336} C_VEL
LIN {X 0,Y 251.886,Z 375.642,A -85,B 0,C 180,E1 -18946.872,E2 -18946.872} C_VEL
LIN {X 0,Y 253.907,Z 379.145,A -85,B 0,C 180,E1 -18947.478,E2 -18947.478} C_VEL
LIN {X 0,Y 259.153,Z 389.014,A -85,B 0,C 180,E1 -18949.167,E2 -18949.167} C_VEL
LIN {X 0,Y 264.161,Z 400.343,A -85,B 0,C 180,E1 -18951.003,E2 -18951.003} C_VEL
LIN {X 0,Y 268.431,Z 412.637,A -85,B 0,C 180,E1 -18952.973,E2 -18952.973} C_VEL
LIN {X 0,Y 271.602,Z 424.935,A -85,B 0,C 180,E1 -18954.962,E2 -18954.962} C_VEL
LIN {X 0,Y 273.049,Z 432.977,A -85,B 0,C 180,E1 -18956.29,E2 -18956.29} C_VEL
LIN {X 0,Y 270.024,Z 446.188,A -85,B 0,C 180,E1 -18957.973,E2 -18957.973} C_VEL
LIN {X 0,Y 266.534,Z 458.786,A -85,B 0,C 180,E1 -18959.934,E2 -18959.934} C_VEL
LIN {X 0,Y 263.305,Z 469.709,A -85,B 0,C 180,E1 -18962.034,E2 -18962.034} C_VEL
LIN {X 0,Y 260.066,Z 479.791,A -85,B 0,C 180,E1 -18964.38,E2 -18964.38} C_VEL
LIN {X 0,Y 256.92,Z 489.189,A -85,B 0,C 180,E1 -18967.057,E2 -18967.057} C_VEL
LIN {X 0,Y 254.222,Z 497.006,A -85,B 0,C 180,E1 -18969.784,E2 -18969.784} C_VEL
LIN {X 0,Y 251.837,Z 504.285,A -85,B 0,C 180,E1 -18972.96,E2 -18972.96} C_VEL
LIN {X 0,Y 249.873,Z 510.06,A -85,B 0,C 180,E1 -18976.167,E2 -18976.167} C_VEL
LIN {X 0,Y 248.877,Z 513.47,A -85,B 0,C 180,E1 -18978.598,E2 -18978.598} C_VEL
LIN {X 0,Y 247.91,Z 516.92,A -85,B 0,C 180,E1 -18981.85,E2 -18981.85} C_VEL
LIN {X 0,Y 247.432,Z 519.192,A -85,B 0,C 180,E1 -18985.111,E2 -18985.111} C_VEL
LIN {X 0,Y 247.167,Z 520.352,A -85,B 0,C 180,E1 -18988.37,E2 -18988.37} C_VEL
LIN {X 0,Y 247.167,Z 520.365,A -85,B 0,C 180,E1 -18991.629,E2 -18991.629} C_VEL
LIN {X 0,Y 247.432,Z 519.256,A -85,B 0,C 180,E1 -18994.887,E2 -18994.887} C_VEL
LIN {X 0,Y 247.908,Z 517.032,A -85,B 0,C 180,E1 -18998.148,E2 -18998.148} C_VEL
LIN {X 0,Y 248.838,Z 513.629,A -85,B 0,C 180,E1 -19001.402,E2 -19001.402} C_VEL
LIN {X 0,Y 250.201,Z 508.965,A -85,B 0,C 180,E1 -19004.643,E2 -19004.643} C_VEL
LIN {X 0,Y 252.31,Z 502.902,A -85,B 0,C 180,E1 -19007.842,E2 -19007.842} C_VEL
LIN {X 0,Y 254.469,Z 496.318,A -85,B 0,C 180,E1 -19010.617,E2 -19010.617} C_VEL
LIN {X 0,Y 257.26,Z 488.34,A -85,B 0,C 180,E1 -19013.335,E2 -19013.335} C_VEL
LIN {X 0,Y 260.448,Z 478.762,A -85,B 0,C 180,E1 -19016.007,E2 -19016.007} C_VEL
LIN {X 0,Y 263.349,Z 469.626,A -85,B 0,C 180,E1 -19018.11,E2 -19018.11} C_VEL
LIN {X 0,Y 266.685,Z 458.35,A -85,B 0,C 180,E1 -19020.265,E2 -19020.265} C_VEL
LIN {X 0,Y 270.211,Z 445.656,A -85,B 0,C 180,E1 -19022.22,E2 -19022.22} C_VEL
LIN {X 0,Y 273.159,Z 433.414,A -85,B 0,C 180,E1 -19023.762,E2 -19023.762} C_VEL
LIN {X 0,Y 271.013,Z 422.137,A -85,B 0,C 180,E1 -19025.631,E2 -19025.631} C_VEL
LIN {X 0,Y 267.517,Z 409.588,A -85,B 0,C 180,E1 -19027.64,E2 -19027.64} C_VEL
LIN {X 0,Y 262.741,Z 396.821,A -85,B 0,C 180,E1 -19029.687,E2 -19029.687} C_VEL
LIN {X 0,Y 257.559,Z 385.766,A -85,B 0,C 180,E1 -19031.523,E2 -19031.523} C_VEL
LIN {X 0,Y 253.761,Z 378.933,A -85,B 0,C 180,E1 -19032.712,E2 -19032.712} C_VEL
LIN {X 0,Y 251.205,Z 374.657,A -85,B 0,C 180,E1 -19033.47,E2 -19033.47} C_VEL
LIN {X 0,Y 249.493,Z 372.135,A -85,B 0,C 180,E1 -19033.967,E2 -19033.967} C_VEL
LIN {X 0,Y 248.992,Z 370.277,A -85,B 0,C 180,E1 -19034.197,E2 -19034.197} C_VEL
LIN {X 0,Y 249.007,Z 370.095,A -85,B 0,C 180,E1 -19037.361,E2 -19037.361} C_VEL
LIN {X 0,Y 249.037,Z 370.089,A -85,B 0,C 180,E1 -19041.621,E2 -19041.621} C_VEL
LIN {X 0,Y 249.06,Z 370.074,A -85,B 0,C 180,E1 -19045.642,E2 -19045.642} C_VEL
LIN {X 0,Y 249.05,Z 370.087,A -85,B 0,C 180,E1 -19049.473,E2 -19049.473} C_VEL
LIN {X 0,Y 249.072,Z 370.06,A -85,B 0,C 180,E1 -19053.162,E2 -19053.162} C_VEL
LIN {X 0,Y 249.078,Z 370.082,A -85,B 0,C 180,E1 -19056.732,E2 -19056.732} C_VEL
LIN {X 0,Y 249.108,Z 370.051,A -85,B 0,C 180,E1 -19060.211,E2 -19060.211} C_VEL
LIN {X 0,Y 249.24,Z 370.062,A -85,B 0,C 180,E1 -19063.622,E2 -19063.622} C_VEL
LIN {X 0,Y 249.252,Z 370.043,A -85,B 0,C 180,E1 -19068.616,E2 -19068.616} C_VEL
LIN {X 0,Y 249.482,Z 370.031,A -85,B 0,C 180,E1 -19071.903,E2 -19071.903} C_VEL
LIN {X 0,Y 249.436,Z 370.039,A -85,B 0,C 180,E1 -19076.769,E2 -19076.769} C_VEL
LIN {X 0,Y 249.734,Z 370.004,A -85,B 0,C 180,E1 -19080,E2 -19080} C_VEL
LIN {X 0,Y 249.436,Z 370.041,A -85,B 0,C 180,E1 -19083.23,E2 -19083.23} C_VEL
LIN {X 0,Y 249.482,Z 370.034,A -85,B 0,C 180,E1 -19088.097,E2 -19088.097} C_VEL
LIN {X 0,Y 249.251,Z 370.062,A -85,B 0,C 180,E1 -19091.383,E2 -19091.383} C_VEL
LIN {X 0,Y 249.24,Z 370.06,A -85,B 0,C 180,E1 -19096.378,E2 -19096.378} C_VEL
LIN {X 0,Y 249.085,Z 370.084,A -85,B 0,C 180,E1 -19101.518,E2 -19101.518} C_VEL
LIN {X 0,Y 249.156,Z 370.41,A -85,B 0,C 180,E1 -19104.679,E2 -19104.679} C_VEL
LIN {X 0,Y 249.605,Z 373.097,A -85,B 0,C 180,E1 -19109.21,E2 -19109.21} C_VEL
LIN {X 0,Y 249.787,Z 374.737,A -85,B 0,C 180,E1 -19111.574,E2 -19111.574} C_VEL
LIN {X 0,Y 249.287,Z 375.814,A -85,B 0,C 180,E1 -19112.902,E2 -19112.902} C_VEL
LIN {X 0,Y 246.696,Z 377.948,A -85,B 0,C 180,E1 -19115.059,E2 -19115.059} C_VEL
LIN {X 0,Y 244.504,Z 379.726,A -85,B 0,C 180,E1 -19116.812,E2 -19116.812} C_VEL
LIN {X 0,Y 243.673,Z 380.967,A -85,B 0,C 180,E1 -19118.171,E2 -19118.171} C_VEL
LIN {X 0,Y 243.668,Z 381.343,A -85,B 0,C 180,E1 -19118.631,E2 -19118.631} C_VEL
LIN {X 0,Y 244.084,Z 383.701,A -85,B 0,C 180,E1 -19121.53,E2 -19121.53} C_VEL
LIN {X 0,Y 244.502,Z 386.689,A -85,B 0,C 180,E1 -19124.819,E2 -19124.819} C_VEL
LIN {X 0,Y 245.49,Z 389.592,A -85,B 0,C 180,E1 -19125.176,E2 -19125.176} C_VEL
LIN {X 0,Y 247.364,Z 392.619,A -85,B 0,C 180,E1 -19125.742,E2 -19125.742} C_VEL
LIN {X 0,Y 251.193,Z 401.199,A -85,B 0,C 180,E1 -19127.038,E2 -19127.038} C_VEL
LIN {X 0,Y 255.475,Z 413.56,A -85,B 0,C 180,E1 -19128.771,E2 -19128.771} C_VEL
LIN {X 0,Y 258.492,Z 424.607,A -85,B 0,C 180,E1 -19130.318,E2 -19130.318} C_VEL
LIN {X 0,Y 261.097,Z 438.296,A -85,B 0,C 180,E1 -19132.249,E2 -19132.249} C_VEL
LIN {X 0,Y 262.554,Z 452.198,A -85,B 0,C 180,E1 -19134.306,E2 -19134.306} C_VEL
LIN {X 0,Y 262.935,Z 464.246,A -85,B 0,C 180,E1 -19136.229,E2 -19136.229} C_VEL
LIN {X 0,Y 259.716,Z 475.866,A -85,B 0,C 180,E1 -19137.924,E2 -19137.924} C_VEL
LIN {X 0,Y 256.122,Z 487.342,A -85,B 0,C 180,E1 -19139.949,E2 -19139.949} C_VEL
LIN {X 0,Y 252.67,Z 497.909,A -85,B 0,C 180,E1 -19142.232,E2 -19142.232} C_VEL
LIN {X 0,Y 249.241,Z 508.258,A -85,B 0,C 180,E1 -19144.979,E2 -19144.979} C_VEL
LIN {X 0,Y 246.344,Z 516.875,A -85,B 0,C 180,E1 -19147.79,E2 -19147.79} C_VEL
LIN {X 0,Y 244.002,Z 524.056,A -85,B 0,C 180,E1 -19150.657,E2 -19150.657} C_VEL
LIN {X 0,Y 242.06,Z 530.736,A -85,B 0,C 180,E1 -19153.99,E2 -19153.99} C_VEL
LIN {X 0,Y 240.745,Z 535.975,A -85,B 0,C 180,E1 -19157.354,E2 -19157.354} C_VEL
LIN {X 0,Y 240.168,Z 539.017,A -85,B 0,C 180,E1 -19159.889,E2 -19159.889} C_VEL
LIN {X 0,Y 239.878,Z 541.992,A -85,B 0,C 180,E1 -19163.271,E2 -19163.271} C_VEL
LIN {X 0,Y 239.926,Z 543.774,A -85,B 0,C 180,E1 -19166.642,E2 -19166.642} C_VEL
LIN {X 0,Y 240.021,Z 544.386,A -85,B 0,C 180,E1 -19170.001,E2 -19170.001} C_VEL
LIN {X 0,Y 239.934,Z 543.762,A -85,B 0,C 180,E1 -19173.359,E2 -19173.359} C_VEL
LIN {X 0,Y 239.959,Z 541.967,A -85,B 0,C 180,E1 -19176.729,E2 -19176.729} C_VEL
LIN {X 0,Y 240.17,Z 538.978,A -85,B 0,C 180,E1 -19180.113,E2 -19180.113} C_VEL
LIN {X 0,Y 241.029,Z 534.747,A -85,B 0,C 180,E1 -19183.49,E2 -19183.49} C_VEL
LIN {X 0,Y 242.59,Z 528.756,A -85,B 0,C 180,E1 -19187.054,E2 -19187.054} C_VEL
LIN {X 0,Y 244.597,Z 522.07,A -85,B 0,C 180,E1 -19190.17,E2 -19190.17} C_VEL
LIN {X 0,Y 247.155,Z 514.509,A -85,B 0,C 180,E1 -19193.017,E2 -19193.017} C_VEL
LIN {X 0,Y 250.288,Z 505.148,A -85,B 0,C 180,E1 -19195.884,E2 -19195.884} C_VEL
LIN {X 0,Y 253.796,Z 494.474,A -85,B 0,C 180,E1 -19198.535,E2 -19198.535} C_VEL
LIN {X 0,Y 257.668,Z 482.202,A -85,B 0,C 180,E1 -19200.986,E2 -19200.986} C_VEL
LIN {X 0,Y 261.354,Z 470.254,A -85,B 0,C 180,E1 -19202.896,E2 -19202.896} C_VEL
LIN {X 0,Y 262.688,Z 465.472,A -85,B 0,C 180,E1 -19203.552,E2 -19203.552} C_VEL
LIN {X 0,Y 262.649,Z 454.92,A -85,B 0,C 180,E1 -19205.24,E2 -19205.24} C_VEL
LIN {X 0,Y 261.703,Z 443.529,A -85,B 0,C 180,E1 -19206.966,E2 -19206.966} C_VEL
LIN {X 0,Y 259.855,Z 431.391,A -85,B 0,C 180,E1 -19208.699,E2 -19208.699} C_VEL
LIN {X 0,Y 256.725,Z 417.832,A -85,B 0,C 180,E1 -19210.584,E2 -19210.584} C_VEL
LIN {X 0,Y 252.967,Z 406.18,A -85,B 0,C 180,E1 -19212.22,E2 -19212.22} C_VEL
LIN {X 0,Y 249.035,Z 396.14,A -85,B 0,C 180,E1 -19213.665,E2 -19213.665} C_VEL
LIN {X 0,Y 247.212,Z 392.123,A -85,B 0,C 180,E1 -19214.255,E2 -19214.255} C_VEL
LIN {X 0,Y 245.046,Z 388.554,A -85,B 0,C 180,E1 -19214.913,E2 -19214.913} C_VEL
LIN {X 0,Y 244.517,Z 386.492,A -85,B 0,C 180,E1 -19215.179,E2 -19215.179} C_VEL
LIN {X 0,Y 244.098,Z 383.598,A -85,B 0,C 180,E1 -19218.532,E2 -19218.532} C_VEL
LIN {X 0,Y 243.509,Z 380.24,A -85,B 0,C 180,E1 -19222.693,E2 -19222.693} C_VEL
LIN {X 0,Y 242.969,Z 376.965,A -85,B 0,C 180,E1 -19227.019,E2 -19227.019} C_VEL
LIN {X 0,Y 242.641,Z 374.633,A -85,B 0,C 180,E1 -19230.502,E2 -19230.502} C_VEL
LIN {X 0,Y 242.31,Z 372.346,A -85,B 0,C 180,E1 -19234.211,E2 -19234.211} C_VEL
LIN {X 0,Y 242.085,Z 371.324,A -85,B 0,C 180,E1 -19236.019,E2 -19236.019} C_VEL
LIN {X 0,Y 242.041,Z 370.961,A -85,B 0,C 180,E1 -19239.608,E2 -19239.608} C_VEL
LIN {X 0,Y 242.167,Z 370.947,A -85,B 0,C 180,E1 -19243.279,E2 -19243.279} C_VEL
LIN {X 0,Y 242.19,Z 370.947,A -85,B 0,C 180,E1 -19248.28,E2 -19248.28} C_VEL
LIN {X 0,Y 242.439,Z 370.914,A -85,B 0,C 180,E1 -19251.666,E2 -19251.666} C_VEL
LIN {X 0,Y 242.265,Z 370.935,A -85,B 0,C 180,E1 -19255.007,E2 -19255.007} C_VEL
LIN {X 0,Y 242.64,Z 370.887,A -85,B 0,C 180,E1 -19258.34,E2 -19258.34} C_VEL
LIN {X 0,Y 242.641,Z 370.886,A -85,B 0,C 180,E1 -19261.66,E2 -19261.66} C_VEL
LIN {X 0,Y 242.435,Z 370.905,A -85,B 0,C 180,E1 -19266.71,E2 -19266.71} C_VEL
LIN {X 0,Y 242.349,Z 370.915,A -85,B 0,C 180,E1 -19270.02,E2 -19270.02} C_VEL
LIN {X 0,Y 242.17,Z 370.932,A -85,B 0,C 180,E1 -19275.141,E2 -19275.141} C_VEL
LIN {X 0,Y 242.075,Z 370.937,A -85,B 0,C 180,E1 -19278.624,E2 -19278.624} C_VEL
LIN {X 0,Y 242.01,Z 370.945,A -85,B 0,C 180,E1 -19282.18,E2 -19282.18} C_VEL
LIN {X 0,Y 242.07,Z 370.939,A -85,B 0,C 180,E1 -19285.838,E2 -19285.838} C_VEL
LIN {X 0,Y 242.011,Z 370.959,A -85,B 0,C 180,E1 -19289.583,E2 -19289.583} C_VEL
LIN {X 0,Y 241.994,Z 370.944,A -85,B 0,C 180,E1 -19293.491,E2 -19293.491} C_VEL
LIN {X 0,Y 242.006,Z 370.966,A -85,B 0,C 180,E1 -19297.579,E2 -19297.579} C_VEL
LIN {X 0,Y 241.941,Z 370.975,A -85,B 0,C 180,E1 -19301.922,E2 -19301.922} C_VEL
LIN {X 0,Y 241.914,Z 370.981,A -85,B 0,C 180,E1 -19304.342,E2 -19304.342} C_VEL
LIN {X 0,Y 242.935,Z 373.855,A -85,B 0,C 180,E1 -19304.741,E2 -19304.741} C_VEL
LIN {X 0,Y 245.044,Z 376.408,A -85,B 0,C 180,E1 -19305.367,E2 -19305.367} C_VEL
LIN {X 0,Y 247.014,Z 379.674,A -85,B 0,C 180,E1 -19305.997,E2 -19305.997} C_VEL
LIN {X 0,Y 251.963,Z 388.453,A -85,B 0,C 180,E1 -19307.661,E2 -19307.661} C_VEL
LIN {X 0,Y 257.589,Z 400.817,A -85,B 0,C 180,E1 -19309.813,E2 -19309.813} C_VEL
LIN {X 0,Y 261.928,Z 413.048,A -85,B 0,C 180,E1 -19311.892,E2 -19311.892} C_VEL
LIN {X 0,Y 265.088,Z 425.138,A -85,B 0,C 180,E1 -19313.942,E2 -19313.942} C_VEL
LIN {X 0,Y 266.803,Z 434.573,A -85,B 0,C 180,E1 -19315.57,E2 -19315.57} C_VEL
LIN {X 0,Y 265.683,Z 439.914,A -85,B 0,C 180,E1 -19316.254,E2 -19316.254} C_VEL
LIN {X 0,Y 262.404,Z 452.557,A -85,B 0,C 180,E1 -19318.064,E2 -19318.064} C_VEL
LIN {X 0,Y 259.159,Z 463.171,A -85,B 0,C 180,E1 -19319.887,E2 -19319.887} C_VEL
LIN {X 0,Y 255.813,Z 473.929,A -85,B 0,C 180,E1 -19322.157,E2 -19322.157} C_VEL
LIN {X 0,Y 252.717,Z 483.051,A -85,B 0,C 180,E1 -19324.465,E2 -19324.465} C_VEL
LIN {X 0,Y 249.515,Z 491.966,A -85,B 0,C 180,E1 -19327.213,E2 -19327.213} C_VEL
LIN {X 0,Y 246.426,Z 500.358,A -85,B 0,C 180,E1 -19330.444,E2 -19330.444} C_VEL
LIN {X 0,Y 244.458,Z 506.225,A -85,B 0,C 180,E1 -19333.291,E2 -19333.291} C_VEL
LIN {X 0,Y 242.564,Z 511.629,A -85,B 0,C 180,E1 -19336.597,E2 -19336.597} C_VEL
LIN {X 0,Y 241.296,Z 515.698,A -85,B 0,C 180,E1 -19339.935,E2 -19339.935} C_VEL
LIN {X 0,Y 240.551,Z 518.614,A -85,B 0,C 180,E1 -19343.391,E2 -19343.391} C_VEL
LIN {X 0,Y 240.229,Z 520.255,A -85,B 0,C 180,E1 -19346.645,E2 -19346.645} C_VEL
LIN {X 0,Y 240.062,Z 520.854,A -85,B 0,C 180,E1 -19349.999,E2 -19349.999} C_VEL
LIN {X 0,Y 240.228,Z 520.293,A -85,B 0,C 180,E1 -19353.354,E2 -19353.354} C_VEL
LIN {X 0,Y 240.571,Z 518.635,A -85,B 0,C 180,E1 -19356.71,E2 -19356.71} C_VEL
LIN {X 0,Y 241.285,Z 515.832,A -85,B 0,C 180,E1 -19360.064,E2 -19360.064} C_VEL
LIN {X 0,Y 242.525,Z 511.809,A -85,B 0,C 180,E1 -19363.404,E2 -19363.404} C_VEL
LIN {X 0,Y 244.399,Z 506.463,A -85,B 0,C 180,E1 -19366.711,E2 -19366.711} C_VEL
LIN {X 0,Y 246.694,Z 499.65,A -85,B 0,C 180,E1 -19369.99,E2 -19369.99} C_VEL
LIN {X 0,Y 249.884,Z 491.12,A -85,B 0,C 180,E1 -19373.187,E2 -19373.187} C_VEL
LIN {X 0,Y 253.096,Z 482.046,A -85,B 0,C 180,E1 -19375.934,E2 -19375.934} C_VEL
LIN {X 0,Y 256.412,Z 472.279,A -85,B 0,C 180,E1 -19378.354,E2 -19378.354} C_VEL
LIN {X 0,Y 259.972,Z 460.812,A -85,B 0,C 180,E1 -19380.68,E2 -19380.68} C_VEL
LIN {X 0,Y 263.598,Z 448.555,A -85,B 0,C 180,E1 -19382.676,E2 -19382.676} C_VEL
LIN {X 0,Y 266.944,Z 435.023,A -85,B 0,C 180,E1 -19384.474,E2 -19384.474} C_VEL
LIN {X 0,Y 264.542,Z 422.395,A -85,B 0,C 180,E1 -19386.659,E2 -19386.659} C_VEL
LIN {X 0,Y 261.101,Z 410.417,A -85,B 0,C 180,E1 -19388.685,E2 -19388.685} C_VEL
LIN {X 0,Y 256.506,Z 398.114,A -85,B 0,C 180,E1 -19390.775,E2 -19390.775} C_VEL
LIN {X 0,Y 251.111,Z 386.787,A -85,B 0,C 180,E1 -19392.794,E2 -19392.794} C_VEL
LIN {X 0,Y 246.831,Z 379.456,A -85,B 0,C 180,E1 -19394.211,E2 -19394.211} C_VEL
LIN {X 0,Y 244.939,Z 376.114,A -85,B 0,C 180,E1 -19394.825,E2 -19394.825} C_VEL
LIN {X 0,Y 242.567,Z 373.214,A -85,B 0,C 180,E1 -19395.536,E2 -19395.536} C_VEL
LIN {X 0,Y 241.895,Z 370.979,A -85,B 0,C 180,E1 -19395.847,E2 -19395.847} C_VEL
LIN {X 0,Y 241.971,Z 370.971,A -85,B 0,C 180,E1 -19400.284,E2 -19400.284} C_VEL
LIN {X 0,Y 242.035,Z 370.962,A -85,B 0,C 180,E1 -19404.497,E2 -19404.497} C_VEL
LIN {X 0,Y 241.975,Z 370.958,A -85,B 0,C 180,E1 -19408.48,E2 -19408.48} C_VEL
LIN {X 0,Y 242.007,Z 370.94,A -85,B 0,C 180,E1 -19412.312,E2 -19412.312} C_VEL
LIN {X 0,Y 242.056,Z 370.959,A -85,B 0,C 180,E1 -19416.016,E2 -19416.016} C_VEL
LIN {X 0,Y 242.035,Z 370.93,A -85,B 0,C 180,E1 -19419.608,E2 -19419.608} C_VEL
LIN {X 0,Y 242.161,Z 370.946,A -85,B 0,C 180,E1 -19423.278,E2 -19423.278} C_VEL
LIN {X 0,Y 242.185,Z 370.918,A -85,B 0,C 180,E1 -19428.28,E2 -19428.28} C_VEL
LIN {X 0,Y 242.433,Z 370.91,A -85,B 0,C 180,E1 -19431.666,E2 -19431.666} C_VEL
LIN {X 0,Y 242.26,Z 370.934,A -85,B 0,C 180,E1 -19435.007,E2 -19435.007} C_VEL
LIN {X 0,Y 242.635,Z 370.887,A -85,B 0,C 180,E1 -19438.34,E2 -19438.34} C_VEL
LIN {X 0,Y 242.635,Z 370.89,A -85,B 0,C 180,E1 -19441.66,E2 -19441.66} C_VEL
LIN {X 0,Y 242.432,Z 370.912,A -85,B 0,C 180,E1 -19446.659,E2 -19446.659} C_VEL
LIN {X 0,Y 242.343,Z 370.922,A -85,B 0,C 180,E1 -19450.02,E2 -19450.02} C_VEL
LIN {X 0,Y 242.165,Z 370.939,A -85,B 0,C 180,E1 -19455.141,E2 -19455.141} C_VEL
LIN {X 0,Y 242.071,Z 370.953,A -85,B 0,C 180,E1 -19458.624,E2 -19458.624} C_VEL
LIN {X 0,Y 242.011,Z 370.966,A -85,B 0,C 180,E1 -19462.18,E2 -19462.18} C_VEL
LIN {X 0,Y 242.108,Z 371.377,A -85,B 0,C 180,E1 -19463.979,E2 -19463.979} C_VEL
LIN {X 0,Y 242.459,Z 373.525,A -85,B 0,C 180,E1 -19467.631,E2 -19467.631} C_VEL
LIN {X 0,Y 242.827,Z 376.071,A -85,B 0,C 180,E1 -19471.546,E2 -19471.546} C_VEL
LIN {X 0,Y 243.365,Z 379.328,A -85,B 0,C 180,E1 -19476.042,E2 -19476.042} C_VEL
LIN {X 0,Y 243.668,Z 381.343,A -85,B 0,C 180,E1 -19478.631,E2 -19478.631} C_VEL
LIN {X 0,Y 243.533,Z 382.216,A -85,B 0,C 180,E1 -19479.502,E2 -19479.502} C_VEL
LIN {X 0,Y 242.606,Z 384.103,A -85,B 0,C 180,E1 -19480.76,E2 -19480.76} C_VEL
LIN {X 0,Y 241.428,Z 386.589,A -85,B 0,C 180,E1 -19481.961,E2 -19481.961} C_VEL
LIN {X 0,Y 240.678,Z 389.577,A -85,B 0,C 180,E1 -19483.074,E2 -19483.074} C_VEL
LIN {X 0,Y 240.943,Z 393.075,A -85,B 0,C 180,E1 -19484.09,E2 -19484.09} C_VEL
LIN {X 0,Y 242.022,Z 395.595,A -85,B 0,C 180,E1 -19484.662,E2 -19484.662} C_VEL
LIN {X 0,Y 243.185,Z 397.857,A -85,B 0,C 180,E1 -19485.076,E2 -19485.076} C_VEL
LIN {X 0,Y 246.292,Z 405.038,A -85,B 0,C 180,E1 -19486.244,E2 -19486.244} C_VEL
LIN {X 0,Y 250.137,Z 416.744,A -85,B 0,C 180,E1 -19488.001,E2 -19488.001} C_VEL
LIN {X 0,Y 253.147,Z 428.73,A -85,B 0,C 180,E1 -19489.772,E2 -19489.772} C_VEL
LIN {X 0,Y 255.389,Z 442.395,A -85,B 0,C 180,E1 -19491.809,E2 -19491.809} C_VEL
LIN {X 0,Y 256.461,Z 455.689,A -85,B 0,C 180,E1 -19493.905,E2 -19493.905} C_VEL
LIN {X 0,Y 256.435,Z 466.509,A -85,B 0,C 180,E1 -19495.729,E2 -19495.729} C_VEL
LIN {X 0,Y 252.582,Z 478.813,A -85,B 0,C 180,E1 -19497.615,E2 -19497.615} C_VEL
LIN {X 0,Y 248.676,Z 490.703,A -85,B 0,C 180,E1 -19499.892,E2 -19499.892} C_VEL
LIN {X 0,Y 245.257,Z 500.723,A -85,B 0,C 180,E1 -19502.248,E2 -19502.248} C_VEL
LIN {X 0,Y 241.902,Z 510.546,A -85,B 0,C 180,E1 -19505.086,E2 -19505.086} C_VEL
LIN {X 0,Y 238.893,Z 518.743,A -85,B 0,C 180,E1 -19507.971,E2 -19507.971} C_VEL
LIN {X 0,Y 236.642,Z 525.543,A -85,B 0,C 180,E1 -19510.933,E2 -19510.933} C_VEL
LIN {X 0,Y 234.749,Z 531.836,A -85,B 0,C 180,E1 -19514.37,E2 -19514.37} C_VEL
LIN {X 0,Y 233.475,Z 536.715,A -85,B 0,C 180,E1 -19517.837,E2 -19517.837} C_VEL
LIN {X 0,Y 232.917,Z 540.308,A -85,B 0,C 180,E1 -19521.323,E2 -19521.323} C_VEL
LIN {X 0,Y 232.838,Z 542.738,A -85,B 0,C 180,E1 -19524.919,E2 -19524.919} C_VEL
LIN {X 0,Y 232.918,Z 543.881,A -85,B 0,C 180,E1 -19528.272,E2 -19528.272} C_VEL
LIN {X 0,Y 232.949,Z 544.039,A -85,B 0,C 180,E1 -19530.001,E2 -19530.001} C_VEL
LIN {X 0,Y 232.919,Z 543.877,A -85,B 0,C 180,E1 -19531.73,E2 -19531.73} C_VEL
LIN {X 0,Y 232.847,Z 542.663,A -85,B 0,C 180,E1 -19535.196,E2 -19535.196} C_VEL
LIN {X 0,Y 232.93,Z 540.272,A -85,B 0,C 180,E1 -19538.678,E2 -19538.678} C_VEL
LIN {X 0,Y 233.477,Z 536.67,A -85,B 0,C 180,E1 -19542.165,E2 -19542.165} C_VEL
LIN {X 0,Y 234.753,Z 531.778,A -85,B 0,C 180,E1 -19545.632,E2 -19545.632} C_VEL
LIN {X 0,Y 236.645,Z 525.459,A -85,B 0,C 180,E1 -19549.068,E2 -19549.068} C_VEL
LIN {X 0,Y 239.279,Z 517.547,A -85,B 0,C 180,E1 -19552.448,E2 -19552.448} C_VEL
LIN {X 0,Y 242.302,Z 509.154,A -85,B 0,C 180,E1 -19555.33,E2 -19555.33} C_VEL
LIN {X 0,Y 245.8,Z 499.053,A -85,B 0,C 180,E1 -19558.15,E2 -19558.15} C_VEL
LIN {X 0,Y 249.322,Z 488.743,A -85,B 0,C 180,E1 -19560.491,E2 -19560.491} C_VEL
LIN {X 0,Y 252.965,Z 477.547,A -85,B 0,C 180,E1 -19562.568,E2 -19562.568} C_VEL
LIN {X 0,Y 256.364,Z 466.475,A -85,B 0,C 180,E1 -19564.246,E2 -19564.246} C_VEL
LIN {X 0,Y 256.408,Z 455.468,A -85,B 0,C 180,E1 -19566.092,E2 -19566.092} C_VEL
LIN {X 0,Y 255.273,Z 441.995,A -85,B 0,C 180,E1 -19568.215,E2 -19568.215} C_VEL
LIN {X 0,Y 253.075,Z 428.58,A -85,B 0,C 180,E1 -19570.209,E2 -19570.209} C_VEL
LIN {X 0,Y 249.615,Z 415.078,A -85,B 0,C 180,E1 -19572.197,E2 -19572.197} C_VEL
LIN {X 0,Y 245.62,Z 403.454,A -85,B 0,C 180,E1 -19573.962,E2 -19573.962} C_VEL
LIN {X 0,Y 242.2,Z 395.805,A -85,B 0,C 180,E1 -19575.22,E2 -19575.22} C_VEL
